					// namnv1104
					Monitor_Production.Pulse_In_2 := TRUE;
					Monitor_Production.Pulse_Out_2 := FALSE;
				END_IF
				// namnv - dieu kien tat tin hieu test vision
				IF GVL.Pro4_.Auto.Vs_On_Off  AND (GVL.Pro4_.Process.DATA_MC_VS = 1) THEN
					IF NOT GVL.Pro4_.Signal_In.T_Vs_detect.Q  THEN
						GVL.Pro4_.Auto.Vs_On_Off := FALSE;
						Pro_MC2_4 := 5;
						GVL.Pro4_.Process.DATA_TOOL_A1_IN_OLD := 0;
					ELSE
						//log
					END_IF
				ELSE
					Pro_MC2_4 := 5;
					GVL.Pro4_.Process.DATA_TOOL_A1_IN_OLD := 0;
				END_IF;
				
			END_IF
		40:	// Pick OK
			IF GVL.Pro4_.Process.DATA_TOOL_A2_OUT  = 2 AND Pick_A4_T2_Finish  THEN
				//GVL.Pro4_.Process.DATA_TOOL_A2_OUT := 2;
				Ton_OK_MC2_4.IN := FALSE;
				Ton_Limit_Test_VS.IN := FALSE;
				GVL.Pro4_.Process.DATA_MC_VS := 0;
				Pro_MC2_4 := 5;
			END_IF	
		50: // Pick NG
			IF GVL.Pro4_.Process.DATA_TOOL_A2_OUT  = 3 AND Pick_A4_T2_Finish  THEN
				//GVL.Pro4_.Process.DATA_TOOL_A2_OUT := 3;
				Ton_OK_MC2_4.IN := FALSE;
				Ton_Limit_Test_VS.IN := FALSE;
				GVL.Pro4_.Process.DATA_MC_VS := 0;
				Pro_MC2_4 := 5;
			END_IF
			
		60: // Pick NG - TS
			IF GVL.Pro4_.Process.DATA_TOOL_A2_OUT  = 4 AND Pick_A4_T2_Finish  THEN
				//GVL.Pro4_.Process.DATA_TOOL_A2_OUT := 3;
				Ton_OK_MC2_4.IN := FALSE;
				Ton_Limit_Test_VS.IN := FALSE;
				GVL.Pro4_.Process.DATA_MC_VS := 0;
				GVL.Pro4_.Process.DATA_TOOL_A1_IN_OLD := 0;
				Pro_MC2_4 := 5;
			END_IF
	END_CASE
END_ACTION

ACTION ACT_GO_Pos_Manual:
{region "1. GO HOME"}
Excute_Run_goHome_A := GVL.RB_A.Manual AND GVL.RB_A.RB_goHome_Comfirm AND GVL.RB_A_.Ready AND NOT GVL.RB_A_.Runing AND
					(GVL.RB_A.M1_goHome OR GVL.RB_A.M2_goHome OR GVL.RB_A.M3_goHome OR GVL.RB_A.M4_goHome );
Excute_Run_goHome_B := GVL.RB_B.Manual AND GVL.RB_B.RB_goHome_Comfirm AND GVL.RB_B_.Ready AND NOT GVL.RB_B_.Runing AND
					(GVL.RB_B.M1_goHome OR GVL.RB_B.M2_goHome OR GVL.RB_B.M3_goHome OR GVL.RB_B.M4_goHome );

IF GVL.RB_A.Manual AND GVL.RB_A.RB_goHome_Comfirm THEN
	GVL.RB_A.COORD := 0;
	IF GVL.RB_A.M1_goHome THEN Pos_run_manual_A.a.a0 := 0; ELSE Pos_run_manual_A.a.a0 := GVL.RB_A_.CUR_X ; END_IF;
	IF GVL.RB_A.M2_goHome THEN Pos_run_manual_A.a.a1 := 0; ELSE Pos_run_manual_A.a.a1 := GVL.RB_A_.CUR_Y ; END_IF;	
	IF GVL.RB_A.M3_goHome THEN Pos_run_manual_A.a.a2 := 0; ELSE Pos_run_manual_A.a.a2 := GVL.RB_A_.CUR_Z ; END_IF;	
	IF GVL.RB_A.M4_goHome THEN Pos_run_manual_A.a.a3 := 0; ELSE Pos_run_manual_A.a.a3 := GVL.RB_A_.CUR_R ; END_IF;	
END_IF

IF GVL.RB_B.Manual AND GVL.RB_B.RB_goHome_Comfirm THEN
	GVL.RB_B.COORD := 0;
	IF GVL.RB_B.M1_goHome THEN Pos_run_manual_B.a.a0 := 0; ELSE Pos_run_manual_B.a.a0 := GVL.RB_B_.CUR_X ; END_IF;	
	IF GVL.RB_B.M2_goHome THEN Pos_run_manual_B.a.a1 := 0; ELSE Pos_run_manual_B.a.a1 := GVL.RB_B_.CUR_Y ; END_IF;	
	IF GVL.RB_B.M3_goHome THEN Pos_run_manual_B.a.a2 := 0; ELSE Pos_run_manual_B.a.a2 := GVL.RB_B_.CUR_Z ; END_IF;	
	IF GVL.RB_B.M4_goHome THEN Pos_run_manual_B.a.a3 := 0; ELSE Pos_run_manual_B.a.a3 := GVL.RB_B_.CUR_R ; END_IF;
END_IF
{endregion}	

// Cai dat bien bao den vi tri muc tieu manual	 
IF (MOVP_A.Done OR MOVL_A.Done) 
AND (ABS(GVL.RB_A_.CUR_X - Pos_run_manual_A.c.X) < delta_position_cor) 
AND (ABS(GVL.RB_A_.CUR_Y - Pos_run_manual_A.c.Y) < delta_position_cor) 
AND (ABS(GVL.RB_A_.CUR_Z - Pos_run_manual_A.c.Z) < delta_position_cor) 
AND (ABS(GVL.RB_A_.CUR_R - Pos_run_manual_A.c.A) < delta_position_cor)
THEN  A_Comp_Man	:= TRUE;  ELSE A_Comp_Man	:= FALSE; END_IF;
IF (MOVP_B.Done OR MOVL_B.Done)  
AND (ABS(GVL.RB_B_.CUR_X - Pos_run_manual_B.c.X) < delta_position_cor) 
AND (ABS(GVL.RB_B_.CUR_Y - Pos_run_manual_B.c.Y) < delta_position_cor) 
AND (ABS(GVL.RB_B_.CUR_Z - Pos_run_manual_B.c.Z) < delta_position_cor) 
AND (ABS(GVL.RB_B_.CUR_R - Pos_run_manual_B.c.A) < delta_position_cor)
THEN  B_Comp_Man	:= TRUE;  ELSE B_Comp_Man	:= FALSE; END_IF;


{region "2. GO WAIT"}
// Jog & Teach
AP_Man_Z_Wait_Go := GVL.RB_A.Manual AND GVL.RB_A.Jog_Point AND GVL.RB_A.Move_Z_Wait AND GVL.RB_A_.Ready AND NOT GVL.RB_A_.Runing AND
						Pos_run_manual_A.c.Z = GVL_1.DATA_RB_A.Z_POS[1];
						IF GVL.RB_A.Move_Z_Wait AND POU_HMI_CONTROL_ROBOT.D_HMI_SCREEN = 21 THEN
							GVL.RB_A.COORD := 1;
							Pos_run_manual_A := POU_MONITOR_ROBOT.RB1_POS;
							Pos_run_manual_A.c.Z := GVL_1.DATA_RB_A.Z_POS[1];
						END_IF;																		
AP_Man_R_Wait_Go := GVL.RB_A.Manual AND GVL.RB_A.Jog_Point AND GVL.RB_A.Move_R_Wait AND GVL.RB_A_.Ready AND NOT GVL.RB_A_.Runing AND
						Pos_run_manual_A.c.A = GVL_1.DATA_RB_A.R_POS[1];
						IF GVL.RB_A.Move_R_Wait AND POU_HMI_CONTROL_ROBOT.D_HMI_SCREEN = 21 THEN
							GVL.RB_A.COORD := 1;
							Pos_run_manual_A := POU_MONITOR_ROBOT.RB1_POS;
							Pos_run_manual_A.c.A := GVL_1.DATA_RB_A.R_POS[1];
						END_IF;	
AP_Man_XY_Wait_Go := GVL.RB_A.Manual AND GVL.RB_A.Jog_Point AND GVL.RB_A.Move_XY_Wait AND GVL.RB_A_.Ready AND NOT GVL.RB_A_.Runing AND
						Pos_run_manual_A.c.X = GVL_1.DATA_RB_A.X_POS[1] AND Pos_run_manual_A.c.Y = GVL_1.DATA_RB_A.Y_POS[1] ;
						IF GVL.RB_A.Move_XY_Wait AND POU_HMI_CONTROL_ROBOT.D_HMI_SCREEN = 21 THEN
							GVL.RB_A.COORD := 1;
							Pos_run_manual_A := POU_MONITOR_ROBOT.RB1_POS;
							Pos_run_manual_A.c.X := GVL_1.DATA_RB_A.X_POS[1];
							Pos_run_manual_A.c.Y := GVL_1.DATA_RB_A.Y_POS[1];
						END_IF;	
/////////////////////////////////////////
Excute_Run_goZ_Wait_B := GVL.RB_B.Manual AND GVL.RB_B.Jog_Point AND GVL.RB_B.Move_Z_Wait AND GVL.RB_B_.Ready AND NOT GVL.RB_B_.Runing AND
						Pos_run_manual_B.c.Z = GVL_1.DATA_RB_B.Z_POS[1];
						IF GVL.RB_B.Move_Z_Wait AND POU_HMI_CONTROL_ROBOT.D_HMI_SCREEN = 31 THEN
							GVL.RB_B.COORD := 1;
							Pos_run_manual_B := POU_MONITOR_ROBOT.RB1_POS;
							Pos_run_manual_B.c.Z := GVL_1.DATA_RB_B.Z_POS[1];
						END_IF;																		
Excute_Run_goR_Wait_B := GVL.RB_B.Manual AND GVL.RB_B.Jog_Point AND GVL.RB_B.Move_R_Wait AND GVL.RB_B_.Ready AND NOT GVL.RB_B_.Runing AND
						Pos_run_manual_B.c.A = GVL_1.DATA_RB_B.R_POS[1];
						IF GVL.RB_B.Move_R_Wait AND POU_HMI_CONTROL_ROBOT.D_HMI_SCREEN = 31 THEN
							GVL.RB_B.COORD := 1;
							Pos_run_manual_B := POU_MONITOR_ROBOT.RB1_POS;
							Pos_run_manual_B.c.A := GVL_1.DATA_RB_B.R_POS[1];
						END_IF;	
Excute_Run_goXY_Wait_B := GVL.RB_B.Manual AND GVL.RB_B.Jog_Point AND GVL.RB_B.Move_XY_Wait AND GVL.RB_B_.Ready AND NOT GVL.RB_B_.Runing AND
						Pos_run_manual_B.c.X = GVL_1.DATA_RB_B.X_POS[1] AND Pos_run_manual_B.c.Y = GVL_1.DATA_RB_B.Y_POS[1] ;
						IF GVL.RB_B.Move_XY_Wait AND POU_HMI_CONTROL_ROBOT.D_HMI_SCREEN = 31 THEN
							GVL.RB_B.COORD := 1;
							Pos_run_manual_B := POU_MONITOR_ROBOT.RB1_POS;
							Pos_run_manual_B.c.X := GVL_1.DATA_RB_B.X_POS[1];
							Pos_run_manual_B.c.Y := GVL_1.DATA_RB_B.Y_POS[1];
						END_IF;	
{endregion}	
{region "3. GO SELECT POS"}
// ROBOT A
	AP_Man_Pos_Go := GVL.RB_A.Manual AND GVL.RB_A.Comfirm_Move AND GVL.RB_A_.Ready AND NOT GVL.RB_A_.Runing AND
							GVL.DW_[10] > 0 AND GVL.DW_[11] > 0 AND GVL.DW_[11] = 3;
	AP_Man_Pos_Go_L := GVL.RB_A.Manual AND GVL.RB_A.Comfirm_Move AND GVL.RB_A_.Ready AND NOT GVL.RB_A_.Runing AND
							GVL.DW_[10] > 0 AND GVL.DW_[11] > 0 AND GVL.DW_[11] = 1;
						IF GVL.RB_A.Comfirm_Move AND POU_HMI_CONTROL_ROBOT.D_HMI_SCREEN = 21 THEN
							GVL.RB_A.COORD := 1;						
							Pos_run_manual_A.c.X:= GVL_1.DATA_RB_A.X_POS[GVL.DW_[10]];
							Pos_run_manual_A.c.Y:= GVL_1.DATA_RB_A.Y_POS[GVL.DW_[10]];
							Pos_run_manual_A.c.Z:= GVL_1.DATA_RB_A.Z_POS[GVL.DW_[10]];
							Pos_run_manual_A.c.A:= GVL_1.DATA_RB_A.R_POS[GVL.DW_[10]];
							GVL.RB_A.Comfirm_Move := FALSE;											 
						END_IF;		
	Other_PosA := Pos_run_manual_A.c.X <> Pos_run_A_Pre.c.X OR Pos_run_manual_A.c.Y <> Pos_run_A_Pre.c.Y 
				  OR Pos_run_manual_A.c.Z <> Pos_run_A_Pre.c.Z OR Pos_run_manual_A.c.A <> Pos_run_A_Pre.c.A;	  											 
	Excute_Run_goPos_A_UpZ := GVL.RB_A.Manual AND GVL.RB_A.Comfirm_Up_Z AND GVL.RB_A_.Ready AND NOT GVL.RB_A_.Runing AND
							GVL.DW_[10] > 0 AND GVL.DW_[11] > 0;
	Excute_Run_goPos_A_UpZ_XY_BF_R := GVL.RB_A.Manual AND GVL.RB_A.Comfirm_Up_Z_XY_BF_R AND GVL.RB_A_.Ready AND NOT GVL.RB_A_.Runing AND
							GVL.DW_[10] > 0 AND GVL.DW_[11] > 0;
	Excute_Run_goPos_A_UpZ_R_BF_XY := GVL.RB_A.Manual AND GVL.RB_A.Comfirm_Up_Z_R_BF_XY AND GVL.RB_A_.Ready AND NOT GVL.RB_A_.Runing AND
							GVL.DW_[10] > 0 AND GVL.DW_[11] > 0;
						IF Excute_Run_goPos_A_UpZ AND POU_HMI_CONTROL_ROBOT.D_HMI_SCREEN = 21 THEN
							GVL.RB_A.COORD := 1;						
							RuningPosA[GVL.DW_[10]] := TRUE;
							mode_Run_GoPosA_manual := 1;	// chi len Z
							Pos_Run_A_Pre := Pos_0;		
							GVL.RB_A.Comfirm_Up_Z := FALSE; 
						ELSE
							IF Excute_Run_goPos_A_UpZ_XY_BF_R AND POU_HMI_CONTROL_ROBOT.D_HMI_SCREEN = 21 THEN
								GVL.RB_A.COORD := 1;						
								RuningPosA[GVL.DW_[10]] := TRUE;
								mode_Run_GoPosA_manual := 2;		// chay XY trc xoay R
								Pos_Run_A_Pre := Pos_0;		
								GVL.RB_A.Comfirm_Up_Z_XY_BF_R := FALSE;
							ELSE
								IF Excute_Run_goPos_A_UpZ_R_BF_XY AND POU_HMI_CONTROL_ROBOT.D_HMI_SCREEN = 21 THEN
									GVL.RB_A.COORD := 1;						
									RuningPosA[GVL.DW_[10]] := TRUE;
									mode_Run_GoPosA_manual := 3;		// xoay R trc XY
									Pos_Run_A_Pre := Pos_0;		
									GVL.RB_A.Comfirm_Up_Z_R_BF_XY := FALSE;
								END_IF; 
							END_IF;	 
						END_IF;	

IF NOT GVL.X[9] THEN
	RuningPosA[GVL.DW_[10]] := FALSE;
	RuningPosB[GVL.DW_[12]]	:= FALSE;	 
END_IF;
						 
IF RuningPosA[GVL.DW_[10]] THEN
	CASE PRO_A[GVL.DW_[10]] OF
			0: 
				Pos_run_manual_A :=  POU_MONITOR_ROBOT.RB1_POS;
				PRO_A[GVL.DW_[10]] := PRO_A[GVL.DW_[10]] + 10;
			10:
				Pos_run_manual_A.c.Z :=  GVL_1.DATA_RB_A.Z_POS[1];
				PRO_A[GVL.DW_[10]] := PRO_A[GVL.DW_[10]] + 10;
			20:
				IF Other_PosA THEN
					CASE GVL.DW_[11] OF
						1: 	excute_run_L_Upz_A := TRUE; 
						3:  AP_Man_UP_Z_Go := TRUE;
					END_CASE
					Pos_Run_A_Pre := Pos_run_manual_A; 
				END_IF
				IF GVL.RB_A_.ERROR OR  NOT GVL.RB_A_.Ready THEN
					RuningPosA[GVL.DW_[10]] := FALSE;
					excute_run_L_Upz_A := FALSE; 
					AP_Man_UP_Z_Go := FALSE;
			    END_IF
			    IF MOVL_A.Done OR MOVP_A.Done THEN
					excute_run_L_Upz_A := FALSE; 
					AP_Man_UP_Z_Go := FALSE;
					IF mode_Run_GoPosA_manual = 1 THEN
						PRO_A[GVL.DW_[10]] := PRO_A[GVL.DW_[10]] + 10;
					ELSE
						IF mode_Run_GoPosA_manual = 2 THEN
							PRO_A[GVL.DW_[10]] := PRO_A[GVL.DW_[10]] + 2;
						ELSE
							IF mode_Run_GoPosA_manual = 3 THEN
								PRO_A[GVL.DW_[10]] := PRO_A[GVL.DW_[10]] + 6;	 
							END_IF;
						END_IF;
					END_IF;
			    END_IF;
			22:
				Pos_run_manual_A.c.X :=  GVL_1.DATA_RB_A.X_POS[GVL.DW_[10]];
				Pos_run_manual_A.c.Y :=  GVL_1.DATA_RB_A.Y_POS[GVL.DW_[10]];	
				Pos_run_manual_A.c.Z :=  GVL.RB_A_.CUR_Z;					 
				Pos_run_manual_A.c.A :=  GVL.RB_A_.CUR_R;		  
				PRO_A[GVL.DW_[10]] := PRO_A[GVL.DW_[10]] + 2; 
			24:
				IF Other_PosA THEN
					CASE GVL.DW_[11] OF
						1: 	excute_run_L_Upz_A := TRUE; 
						3:  AP_Man_UP_Z_Go := TRUE;
					END_CASE
					Pos_Run_A_Pre := Pos_run_manual_A; 
				END_IF
				IF GVL.RB_A_.ERROR OR  NOT GVL.RB_A_.Ready THEN
					RuningPosA[GVL.DW_[10]] := FALSE;
					excute_run_L_Upz_A := FALSE; 
					AP_Man_UP_Z_Go := FALSE;
			    END_IF
			    IF MOVL_A.Done OR MOVP_A.Done THEN
					excute_run_L_Upz_A := FALSE; 
					AP_Man_UP_Z_Go := FALSE;
					PRO_A[GVL.DW_[10]] := 30;
			    END_IF	
			26:
				Pos_run_manual_A.c.X :=  GVL.RB_A_.CUR_X;
				Pos_run_manual_A.c.Y :=  GVL.RB_A_.CUR_Y;	
				Pos_run_manual_A.c.Z :=  GVL.RB_A_.CUR_Z;					 
				Pos_run_manual_A.c.A :=  GVL_1.DATA_RB_A.R_POS[GVL.DW_[10]];		  
				PRO_A[GVL.DW_[10]] := PRO_A[GVL.DW_[10]] + 2; 
			28:
				IF Other_PosA THEN
					CASE GVL.DW_[11] OF
						1: 	excute_run_L_Upz_A := TRUE; 
						3:  AP_Man_UP_Z_Go := TRUE;
					END_CASE
					Pos_Run_A_Pre := Pos_run_manual_A; 
				END_IF
				IF GVL.RB_A_.ERROR OR  NOT GVL.RB_A_.Ready THEN
					RuningPosA[GVL.DW_[10]] := FALSE;
					excute_run_L_Upz_A := FALSE; 
					AP_Man_UP_Z_Go := FALSE;
			    END_IF
			    IF MOVL_A.Done OR MOVP_A.Done THEN
					excute_run_L_Upz_A := FALSE; 
					AP_Man_UP_Z_Go := FALSE;
					PRO_A[GVL.DW_[10]] := 30;
			    END_IF 
			30:
				Pos_run_manual_A.c.X :=  GVL_1.DATA_RB_A.X_POS[GVL.DW_[10]];
				Pos_run_manual_A.c.Y :=  GVL_1.DATA_RB_A.Y_POS[GVL.DW_[10]];	
				Pos_run_manual_A.c.Z :=  GVL.RB_A_.CUR_Z;					 
				Pos_run_manual_A.c.A :=  GVL_1.DATA_RB_A.R_POS[GVL.DW_[10]];		  
				PRO_A[GVL.DW_[10]] := PRO_A[GVL.DW_[10]] + 10; 
			40:
				IF Other_PosA THEN
					CASE GVL.DW_[11] OF
						1: 	excute_run_L_Upz_A := TRUE; 
						3:  AP_Man_UP_Z_Go := TRUE;
					END_CASE
					Pos_Run_A_Pre := Pos_run_manual_A; 
				END_IF
				IF GVL.RB_A_.ERROR OR  NOT GVL.RB_A_.Ready THEN
					RuningPosA[GVL.DW_[10]] := FALSE;
					excute_run_L_Upz_A := FALSE; 
					AP_Man_UP_Z_Go := FALSE;
			    END_IF
			    IF MOVL_A.Done OR MOVP_A.Done THEN
					excute_run_L_Upz_A := FALSE; 
					AP_Man_UP_Z_Go := FALSE;
					PRO_A[GVL.DW_[10]] := PRO_A[GVL.DW_[10]] + 10;
			    END_IF	
			50:
				Pos_run_manual_A :=  POU_MONITOR_ROBOT.RB1_POS;
				PRO_A[GVL.DW_[10]] := PRO_A[GVL.DW_[10]] + 10;			 
			60:
				Pos_run_manual_A.c.Z :=  GVL_1.DATA_RB_A.Z_POS[GVL.DW_[10]];
				PRO_A[GVL.DW_[10]] := PRO_A[GVL.DW_[10]] + 10;
			70:
				IF Other_PosA THEN
					CASE GVL.DW_[11] OF
						1: 	excute_run_L_Upz_A := TRUE; 
						3:  AP_Man_UP_Z_Go := TRUE;
					END_CASE
					Pos_Run_A_Pre := Pos_run_manual_A; 
				END_IF
				IF GVL.RB_A_.ERROR OR  NOT GVL.RB_A_.Ready THEN
					RuningPosA[GVL.DW_[10]] := FALSE;
					excute_run_L_Upz_A := FALSE; 
					AP_Man_UP_Z_Go := FALSE;
			    END_IF
			    IF MOVL_A.Done OR MOVP_A.Done THEN
					excute_run_L_Upz_A := FALSE; 
					AP_Man_UP_Z_Go := FALSE;
					PRO_A[GVL.DW_[10]] := PRO_A[GVL.DW_[10]] + 10;
			    END_IF			  		   							 
											  
			80:/// HOÀN THÀNH ///  	   
					excute_run_L_Upz_A := FALSE; 
					AP_Man_UP_Z_Go := FALSE;
 			        RuningPosA[GVL.DW_[10]] := FALSE;				
					mode_Run_GoPosA_manual := 0; 
		 END_CASE
ELSE
	PRO_A[GVL.DW_[10]] := 0;	
	excute_run_L_Upz_A := FALSE; 
	AP_Man_UP_Z_Go := FALSE;
	mode_Run_GoPosA_manual := 0; 
END_IF;							  
// ROBOT B
	Excute_Run_goPos_B := GVL.RB_B.Manual AND GVL.RB_B.Comfirm_Move AND GVL.RB_B_.Ready AND NOT GVL.RB_B_.Runing AND
							GVL.DW_[12] > 0 AND GVL.DW_[13] > 0 AND GVL.DW_[13] = 3;
	Excute_Run_goPos_B_L := GVL.RB_B.Manual AND GVL.RB_B.Comfirm_Move AND GVL.RB_B_.Ready AND NOT GVL.RB_B_.Runing AND
							GVL.DW_[12] > 0 AND GVL.DW_[13] > 0 AND GVL.DW_[13] = 1;
							
						IF GVL.RB_B.Comfirm_Move AND POU_HMI_CONTROL_ROBOT.D_HMI_SCREEN = 31 THEN
							GVL.RB_B.COORD := 1;						
							Pos_run_manual_B.c.X:= GVL_1.DATA_RB_B.X_POS[GVL.DW_[12]];
							Pos_run_manual_B.c.Y:= GVL_1.DATA_RB_B.Y_POS[GVL.DW_[12]];
							Pos_run_manual_B.c.Z:= GVL_1.DATA_RB_B.Z_POS[GVL.DW_[12]];
							Pos_run_manual_B.c.A:= GVL_1.DATA_RB_B.R_POS[GVL.DW_[12]];
							GVL.RB_B.Comfirm_Move := FALSE;											 
						END_IF;		
	Other_PosB := Pos_run_manual_B.c.X <> Pos_Run_B_Pre.c.X OR Pos_run_manual_B.c.Y <> Pos_Run_B_Pre.c.Y 
				  OR Pos_run_manual_B.c.Z <> Pos_Run_B_Pre.c.Z OR Pos_run_manual_B.c.A <> Pos_Run_B_Pre.c.A;	  											 
	Excute_Run_goPos_B_UpZ := GVL.RB_B.Manual AND GVL.RB_B.Comfirm_Up_Z AND GVL.RB_B_.Ready AND NOT GVL.RB_B_.Runing AND
							GVL.DW_[12] > 0 AND GVL.DW_[13] > 0;
	Excute_Run_goPos_B_UpZ_XY_BF_R := GVL.RB_B.Manual AND GVL.RB_B.Comfirm_Up_Z_XY_BF_R AND GVL.RB_B_.Ready AND NOT GVL.RB_B_.Runing AND
							GVL.DW_[12] > 0 AND GVL.DW_[13] > 0;
	Excute_Run_goPos_B_UpZ_R_BF_XY := GVL.RB_B.Manual AND GVL.RB_B.Comfirm_Up_Z_R_BF_XY AND GVL.RB_B_.Ready AND NOT GVL.RB_B_.Runing AND
							GVL.DW_[12] > 0 AND GVL.DW_[13] > 0;
						IF Excute_Run_goPos_B_UpZ AND POU_HMI_CONTROL_ROBOT.D_HMI_SCREEN = 31 THEN
							GVL.RB_B.COORD := 1;						
							RuningPosB[GVL.DW_[12]] := TRUE;
							mode_Run_GoPosB_manual := 1;	
							Pos_Run_B_Pre := Pos_0;	
							GVL.RB_B.Comfirm_Up_Z := FALSE;
						ELSE
							IF Excute_Run_goPos_B_UpZ_XY_BF_R AND POU_HMI_CONTROL_ROBOT.D_HMI_SCREEN = 31 THEN
								GVL.RB_B.COORD := 1;						
								RuningPosB[GVL.DW_[12]] := TRUE;
								mode_Run_GoPosB_manual := 2;	
								Pos_Run_B_Pre := Pos_0;	
								GVL.RB_B.Comfirm_Up_Z_XY_BF_R := FALSE;	 
							ELSE
								IF Excute_Run_goPos_B_UpZ_R_BF_XY AND POU_HMI_CONTROL_ROBOT.D_HMI_SCREEN = 31 THEN
									GVL.RB_B.COORD := 1;						
									RuningPosB[GVL.DW_[12]] := TRUE;
									mode_Run_GoPosB_manual := 3;	
									Pos_Run_B_Pre := Pos_0;	
									GVL.RB_B.Comfirm_Up_Z_R_BF_XY := FALSE;
								 END_IF;
							END_IF;
						END_IF;							 
IF RuningPosB[GVL.DW_[12]] THEN
	CASE PRO_B[GVL.DW_[12]] OF
			0: 
				Pos_run_manual_B :=  POU_MONITOR_ROBOT.RB2_POS;
				PRO_B[GVL.DW_[12]] := PRO_B[GVL.DW_[12]] + 10;
			10:
				Pos_run_manual_B.c.Z :=  GVL_1.DATA_RB_B.Z_POS[1];
				PRO_B[GVL.DW_[12]] := PRO_B[GVL.DW_[12]] + 10;
			20:
				IF Other_PosB THEN
					CASE GVL.DW_[13] OF
						1: 	excute_run_L_Upz_B := TRUE; 
						3:  excute_run_P_Upz_B := TRUE;
					END_CASE
					Pos_Run_B_Pre := Pos_run_manual_B; 
				END_IF
				IF GVL.RB_B_.ERROR OR  NOT GVL.RB_B_.Ready THEN
					RuningPosB[GVL.DW_[12]] := FALSE;
					excute_run_L_Upz_B := FALSE; 
					excute_run_P_Upz_B := FALSE;
			    END_IF
			    IF MOVL_B.Done OR MOVP_B.Done THEN
					excute_run_L_Upz_B := FALSE; 
					excute_run_P_Upz_B := FALSE;
					IF mode_Run_GoPosB_manual = 1 THEN
						PRO_B[GVL.DW_[12]] := PRO_B[GVL.DW_[12]] + 10;
					ELSE
						IF mode_Run_GoPosB_manual = 2 THEN
							PRO_B[GVL.DW_[12]] := PRO_B[GVL.DW_[12]] + 2;
						ELSE
							IF mode_Run_GoPosB_manual = 3 THEN
								PRO_B[GVL.DW_[12]] := PRO_B[GVL.DW_[12]] + 6;	 
							END_IF;
						END_IF;
					END_IF;
			    END_IF
			22:
				Pos_run_manual_B.c.X :=  GVL_1.DATA_RB_B.X_POS[GVL.DW_[12]];
				Pos_run_manual_B.c.Y :=  GVL_1.DATA_RB_B.Y_POS[GVL.DW_[12]];	
				Pos_run_manual_B.c.Z :=  GVL.RB_B_.CUR_Z;					 
				Pos_run_manual_B.c.A :=  GVL.RB_B_.CUR_R;		  
				PRO_B[GVL.DW_[12]] := PRO_B[GVL.DW_[12]] + 2;  
			24:
				IF Other_PosB THEN
					CASE GVL.DW_[13] OF
						1: 	excute_run_L_Upz_B := TRUE; 
						3:  excute_run_P_Upz_B := TRUE;
					END_CASE
					Pos_Run_B_Pre := Pos_run_manual_B; 
				END_IF
				IF GVL.RB_B_.ERROR OR NOT GVL.RB_B_.Ready THEN
					RuningPosB[GVL.DW_[12]] := FALSE;
					excute_run_L_Upz_B := FALSE; 
					excute_run_P_Upz_B := FALSE;
			    END_IF
			    IF MOVL_B.Done OR MOVP_B.Done THEN
					excute_run_L_Upz_B := FALSE; 
					excute_run_P_Upz_B := FALSE;
					PRO_B[GVL.DW_[12]] := 30;
			    END_IF
			26:
				Pos_run_manual_B.c.X :=  GVL.RB_B_.CUR_X;
				Pos_run_manual_B.c.Y :=  GVL.RB_B_.CUR_Y;	
				Pos_run_manual_B.c.Z :=  GVL.RB_B_.CUR_Z;					 
				Pos_run_manual_B.c.A :=  GVL_1.DATA_RB_B.r_POS[GVL.DW_[12]];		  
				PRO_B[GVL.DW_[12]] := PRO_B[GVL.DW_[12]] + 2;
			28:
				IF Other_PosB THEN
					CASE GVL.DW_[13] OF
						1: 	excute_run_L_Upz_B := TRUE; 
						3:  excute_run_P_Upz_B := TRUE;
					END_CASE
					Pos_Run_B_Pre := Pos_run_manual_B; 
				END_IF
				IF GVL.RB_B_.ERROR OR NOT GVL.RB_B_.Ready THEN
					RuningPosB[GVL.DW_[12]] := FALSE;
					excute_run_L_Upz_B := FALSE; 
					excute_run_P_Upz_B := FALSE;
			    END_IF
			    IF MOVL_B.Done OR MOVP_B.Done THEN
					excute_run_L_Upz_B := FALSE; 
					excute_run_P_Upz_B := FALSE;
					PRO_B[GVL.DW_[12]] := 30;
			    END_IF 
			30:
				Pos_run_manual_B.c.X :=  GVL_1.DATA_RB_B.X_POS[GVL.DW_[12]];
				Pos_run_manual_B.c.Y :=  GVL_1.DATA_RB_B.Y_POS[GVL.DW_[12]];	
				Pos_run_manual_B.c.Z :=  GVL.RB_B_.CUR_Z;					 
				Pos_run_manual_B.c.A :=  GVL_1.DATA_RB_B.r_POS[GVL.DW_[12]];		  
				PRO_B[GVL.DW_[12]] := PRO_B[GVL.DW_[12]] + 10; 
			40:
				IF Other_PosB THEN
					CASE GVL.DW_[13] OF
						1: 	excute_run_L_Upz_B := TRUE; 
						3:  excute_run_P_Upz_B := TRUE;
					END_CASE
					Pos_Run_B_Pre := Pos_run_manual_B; 
				END_IF
				IF GVL.RB_B_.ERROR OR NOT GVL.RB_B_.Ready THEN
					RuningPosB[GVL.DW_[12]] := FALSE;
					excute_run_L_Upz_B := FALSE; 
					excute_run_P_Upz_B := FALSE;
			    END_IF
			    IF MOVL_B.Done OR MOVP_B.Done THEN
					excute_run_L_Upz_B := FALSE; 
					excute_run_P_Upz_B := FALSE;
					PRO_B[GVL.DW_[12]] := PRO_B[GVL.DW_[12]] + 10;
			    END_IF
			50:
				Pos_run_manual_B :=  POU_MONITOR_ROBOT.RB2_POS;
				PRO_B[GVL.DW_[12]] := PRO_B[GVL.DW_[12]] + 10;			 
			60:
				Pos_run_manual_B.c.Z :=  GVL_1.DATA_RB_B.Z_POS[GVL.DW_[12]];
				PRO_B[GVL.DW_[12]] := PRO_B[GVL.DW_[12]] + 10;
			70:
				IF Other_PosB THEN
					CASE GVL.DW_[13] OF
						1: 	excute_run_L_Upz_B := TRUE; 
						3:  excute_run_P_Upz_B := TRUE;
					END_CASE
					Pos_Run_B_Pre := Pos_run_manual_B; 
				END_IF
				IF GVL.RB_B_.ERROR OR  NOT GVL.RB_b_.Ready THEN
					RuningPosB[GVL.DW_[12]] := FALSE;
					excute_run_L_Upz_B := FALSE; 
					excute_run_P_Upz_B := FALSE;
			    END_IF
			    IF MOVL_B.Done OR MOVP_B.Done THEN
					excute_run_L_Upz_B := FALSE; 
					excute_run_P_Upz_B := FALSE;
					PRO_B[GVL.DW_[12]] := PRO_B[GVL.DW_[12]] + 10;
			    END_IF	
			80:/// HOÀN THÀNH ///  	   
					excute_run_L_Upz_B := FALSE; 
					excute_run_P_Upz_B := FALSE;
 			        RuningPosB[GVL.DW_[12]] := FALSE;			
					mode_Run_GoPosB_manual := 0;	 
		 END_CASE
ELSE
	PRO_B[GVL.DW_[12]] := 0;	
	excute_run_L_Upz_b := FALSE; 
	excute_run_P_Upz_b := FALSE;		
	mode_Run_GoPosB_manual := 0;	 
END_IF;										   
{endregion}	
	 
{region "4. Pos Cam"}	 
// excute_run_cam_B := GVL.RB_B.Manual AND GVL.RB_B_.Ready AND NOT GVL.RB_B_.Runing AND GVL.RB_B.move_Pos_cam ;
// 	 					 
// 						IF GVL.RB_B.move_Pos_cam AND POU_HMI_CONTROL_ROBOT.D_HMI_SCREEN = 31 THEN
// 							GVL.RB_B.COORD := 1;
// 							Pos_run_manual_B := POU_MONITOR_ROBOT.RB1_POS;
// 							Pos_run_manual_B.c.X := GVL_1.DATA_RB_B.X_POS[1];
// 							Pos_run_manual_B.c.Y := GVL_1.DATA_RB_B.Y_POS[1];
// 						END_IF;		  
// ROBOT B
	excute_run_cam_B := GVL.RB_B.Manual AND GVL.RB_B_.Ready AND NOT GVL.RB_B_.Runing AND GVL.RB_B.move_Pos_cam ;	
	  											 
						IF excute_run_cam_B AND POU_HMI_CONTROL_ROBOT.D_HMI_SCREEN = 181 THEN
							GVL.RB_B.COORD := 1;						
							Running_B_Cam := TRUE;	
							Pos_Run_B_Pre := Pos_0;	
							excute_run_cam_B := FALSE;	 
						END_IF;							 
IF Running_B_Cam THEN
	CASE Pro_B_cam OF
			0: 
				Pos_run_manual_B :=  POU_MONITOR_ROBOT.RB2_POS;
				Pro_B_cam := Pro_B_cam + 10;
			10:
				Pos_run_manual_B.c.Z :=  GVL_1.DATA_RB_B.Z_POS[1];
				Pro_B_cam := Pro_B_cam + 10;
			20:
				IF Other_PosB THEN
				excute_run_P_cam_B := TRUE;
				Pos_Run_B_Pre := Pos_run_manual_B; 
				END_IF;
				IF GVL.RB_B_.ERROR OR  NOT GVL.RB_B_.Ready THEN
					excute_run_P_cam_B := FALSE;
				    Running_B_Cam := FALSE;
			    END_IF
			    IF MOVP_B.Done THEN
					excute_run_P_cam_B := FALSE;
					Pro_B_cam := Pro_B_cam + 10;
			    END_IF
			30:
				CASE GVL.DW_[20] OF
					0:
						Pos_run_manual_B.c.X :=  GVL.Cam_T1.POS_X_RESULT;
						Pos_run_manual_B.c.Y :=  GVL.Cam_T1.POS_Y_RESULT;	  					 
					1:	 
						Pos_run_manual_B.c.X :=  GVL.Cam_T2.POS_X_RESULT;
						Pos_run_manual_B.c.Y :=  GVL.Cam_T2.POS_Y_RESULT;	 
				END_CASE		  
						Pos_run_manual_B.c.Z :=  GVL.RB_B_.CUR_Z;					 
						Pos_run_manual_B.c.A :=  GVL_1.DATA_RB_B.r_POS[1];					   
				Pro_B_cam := Pro_B_cam + 10;
			40:
				IF Other_PosB THEN
				excute_run_P_cam_B := TRUE;
				Pos_Run_B_Pre := Pos_run_manual_B; 
				END_IF;
				IF GVL.RB_B_.ERROR OR  NOT GVL.RB_B_.Ready THEN
					excute_run_P_cam_B := FALSE;
				    Running_B_Cam := FALSE;
			    END_IF
			    IF MOVP_B.Done THEN
					excute_run_P_cam_B := FALSE;
					Pro_B_cam := Pro_B_cam + 10;
			    END_IF			 
			50:
				GVL.RB_B.COORD := 1;
				Pos_run_manual_B :=  POU_MONITOR_ROBOT.RB2_POS;
				Pro_B_cam := Pro_B_cam + 10;		 
			60:
				Pos_run_manual_B.c.Z :=  GVL_1.DATA_RB_B.Z_POS[1];
				Pro_B_cam := Pro_B_cam + 10;
			70:
				IF Other_PosB THEN
				excute_run_P_cam_B := TRUE;
				Pos_Run_B_Pre := Pos_run_manual_B; 
				END_IF;
				IF GVL.RB_B_.ERROR OR  NOT GVL.RB_B_.Ready THEN
					excute_run_P_cam_B := FALSE;
				    Running_B_Cam := FALSE;
			    END_IF
			    IF MOVP_B.Done THEN
					excute_run_P_cam_B := FALSE;
					Pro_B_cam := Pro_B_cam + 10;
			    END_IF
			80:/// HOÀN THÀNH ///  	   
					excute_run_P_cam_B:= FALSE; 
 			        Running_B_Cam := FALSE;				 
		 END_CASE
ELSE
	Pro_B_cam := 0;	 
	excute_run_P_cam_B := FALSE;		 
END_IF;			   
/// Test Pick by Cam						
	  											 
IF GVL.MB_[11]  THEN
	CASE Test_Pick OF
			0: 
				Pos_run_manual_B :=  POU_MONITOR_ROBOT.RB2_POS;
				Test_Pick := Test_Pick + 10;
			10:
				Pos_run_manual_B.c.Z :=  GVL_1.DATA_RB_B.Z_POS[1];
				Test_Pick := Test_Pick + 10;
			20:
				IF Other_PosB THEN
				run_P_cam_B_test_pick := TRUE;
				Pos_Run_B_Pre := Pos_run_manual_B; 
				END_IF;
				IF GVL.RB_B_.ERROR OR  NOT GVL.RB_B_.Ready THEN
					run_P_cam_B_test_pick := FALSE;
				    GVL.MB_[11] := FALSE;
			    END_IF
			    IF MOVP_B.Done THEN
					run_P_cam_B_test_pick := FALSE;
					Test_Pick := Test_Pick + 10;
			    END_IF
			30:
				 CASE GVL.DW_[20] OF
					0:
						Pos_run_manual_B.c.X :=  GVL.Cam_T1.POS_X_RESULT;
						Pos_run_manual_B.c.Y :=  GVL.Cam_T1.POS_Y_RESULT;					
					1:	  
						Pos_run_manual_B.c.X :=  GVL.Cam_T2.POS_X_RESULT;
						Pos_run_manual_B.c.Y :=  GVL.Cam_T2.POS_Y_RESULT;						 							  
				 END_CASE	  
				Pos_run_manual_B.c.Z :=  GVL.RB_B_.CUR_Z;					 
				Pos_run_manual_B.c.A :=  GVL_1.DATA_RB_B.r_POS[1];	
// 					 IF GVL.Cam_T2.POS_R_RESULT < 180 THEN
// 						Pos_run_manual_B.c.A:= GVL_1.DATA_RB_B.R_POS[1] + GVL.Cam_T2.POS_R_RESULT ;	  
// 					ELSE
// 						Pos_run_manual_B.c.A:= GVL_1.DATA_RB_B.R_POS[1] - (360-GVL.Cam_T2.POS_R_RESULT) ;	 
// 					END_IF	  
				Test_Pick := Test_Pick + 10;
			40:
				IF Other_PosB THEN
				run_P_cam_B_test_pick := TRUE;
				Pos_Run_B_Pre := Pos_run_manual_B; 
				END_IF;
				IF GVL.RB_B_.ERROR OR  NOT GVL.RB_B_.Ready THEN
					run_P_cam_B_test_pick := FALSE;
				    GVL.MB_[11] := FALSE;
			    END_IF
			    IF MOVP_B.Done THEN
					run_P_cam_B_test_pick := FALSE;
					Test_Pick := Test_Pick + 10;
			    END_IF
			50:
				Pos_run_manual_B :=  POU_MONITOR_ROBOT.RB2_POS;
				Test_Pick := Test_Pick + 10;		 
			60:
				Pos_run_manual_B.c.Z :=  GVL_1.DATA_RB_B.Z_POS[1];
				Test_Pick := Test_Pick + 10;
			70:
				IF Other_PosB THEN
				run_P_cam_B_test_pick := TRUE;
				Pos_Run_B_Pre := Pos_run_manual_B; 
				END_IF;
				IF GVL.RB_B_.ERROR OR  NOT GVL.RB_B_.Ready THEN
					run_P_cam_B_test_pick := FALSE;
				    GVL.MB_[11] := FALSE;
			    END_IF
			    IF MOVP_B.Done THEN
					run_P_cam_B_test_pick := FALSE;
					Test_Pick := Test_Pick + 10;
			    END_IF
			80:	
				 CASE GVL.RB_B.Number_Tool OF
					1:
						GVL.RB_B.Vacuum_1 := TRUE;				
					2:	  
						GVL.RB_B.Vacuum_2 := TRUE;						 							  
				 END_CASE					 
					//Project_3_Delay_A(IN:= TRUE, PT := T#500MS);
				IF Project_3_Delay_A.Q THEN
					Test_Pick := Test_Pick + 10;	
				END_IF;						  
			90: 
				Project_3_Delay_A.IN	:= FALSE;
				Pos_run_manual_B :=  POU_MONITOR_ROBOT.RB2_POS;
				Test_Pick := Test_Pick + 10;
			100:
				Pos_run_manual_B.c.Z :=  GVL_1.DATA_RB_B.Z_POS[1];
				Test_Pick := Test_Pick + 10;
			110:
				IF Other_PosB THEN
				run_P_cam_B_test_pick := TRUE;
				Pos_Run_B_Pre := Pos_run_manual_B; 
				END_IF;
				IF GVL.RB_B_.ERROR OR  NOT GVL.RB_B_.Ready THEN
					run_P_cam_B_test_pick := FALSE;
				    GVL.MB_[11] := FALSE;
			    END_IF
			    IF MOVP_B.Done THEN
					run_P_cam_B_test_pick := FALSE;
					Test_Pick := Test_Pick + 10;
			    END_IF	
			120:
				Pos_run_manual_B.c.X:= GVL_1.DATA_RB_B.X_POS[1];
				Pos_run_manual_B.c.Y:= GVL_1.DATA_RB_B.Y_POS[1];
				Pos_run_manual_B.c.Z:= GVL.RB_B_.CUR_Z;
				Pos_run_manual_B.c.A:= GVL_1.DATA_RB_B.R_POS[1];				 
				Test_Pick := Test_Pick + 10;
			130:
				IF Other_PosB THEN
				run_P_cam_B_test_pick := TRUE;
				Pos_Run_B_Pre := Pos_run_manual_B; 
				END_IF;
				IF GVL.RB_B_.ERROR OR  NOT GVL.RB_B_.Ready THEN
					run_P_cam_B_test_pick := FALSE;
				    GVL.MB_[11] := FALSE;
			    END_IF
			    IF MOVP_B.Done THEN
					run_P_cam_B_test_pick := FALSE;
					Test_Pick := Test_Pick + 10;
			    END_IF						   
			140:/// HOÀN THÀNH ///  	   
					run_P_cam_B_test_pick:= FALSE; 
 			        GVL.MB_[11] := FALSE;			 
		 END_CASE	 
ELSE
run_P_cam_B_test_pick:= FALSE;		 
Test_Pick := 0;			  
END_IF;							 

IF GVL.MB_[12]  THEN
	CASE Test_Place OF
			0: 
				Pos_run_manual_B :=  POU_MONITOR_ROBOT.RB2_POS;
				test_Place := test_Place + 10;
			10:
				Pos_run_manual_B.c.Z :=  GVL_1.DATA_RB_B.Z_POS[1];
				test_Place := test_Place + 10;
			20:
				IF Other_PosB THEN
				run_P_cam_B_test_Place := TRUE;
				Pos_Run_B_Pre := Pos_run_manual_B; 
				END_IF;
				IF GVL.RB_B_.ERROR OR  NOT GVL.RB_B_.Ready THEN
					run_P_cam_B_test_Place := FALSE;
				    GVL.MB_[12] := FALSE;
			    END_IF
			    IF MOVP_B.Done THEN
					run_P_cam_B_test_Place := FALSE;
					test_Place := test_Place + 10;
			    END_IF
			30:
				Pos_run_manual_B.c.X:= GVL_1.DATA_RB_B.X_POS[2];
				Pos_run_manual_B.c.Y:= GVL_1.DATA_RB_B.Y_POS[2];
				Pos_run_manual_B.c.Z:= GVL.RB_B_.CUR_Z;
				Pos_run_manual_B.c.A:= GVL_1.DATA_RB_B.R_POS[2];	 
// 				 CASE GVL.DW_[20] OF
// 					0:
// 						 IF GVL.Cam_T1.POS_R_RESULT < 0 THEN
// 							Pos_run_manual_B.c.A:= GVL_1.DATA_RB_B.R_POS[2] - GVL.Cam_T1.POS_R_RESULT ;	  
// 						ELSE
// 							Pos_run_manual_B.c.A:= GVL_1.DATA_RB_B.R_POS[2] + GVL.Cam_T1.POS_R_RESULT ;	 
// 						END_IF					
// 					1:	  
// 						 IF GVL.Cam_T2.POS_R_RESULT < 0 THEN
// 							Pos_run_manual_B.c.A:= GVL_1.DATA_RB_B.R_POS[2] - GVL.Cam_T2.POS_R_RESULT ;	  
// 						ELSE
// 							Pos_run_manual_B.c.A:= GVL_1.DATA_RB_B.R_POS[2] + GVL.Cam_T2.POS_R_RESULT ;	 
// 						END_IF						 							  
// 				 END_CASE					  
				test_Place := test_Place + 10;
			40:
				IF Other_PosB THEN
				run_P_cam_B_test_Place := TRUE;
				Pos_Run_B_Pre := Pos_run_manual_B; 
				END_IF;
				IF GVL.RB_B_.ERROR OR  NOT GVL.RB_B_.Ready THEN
					run_P_cam_B_test_Place := FALSE;
				    GVL.MB_[12] := FALSE;
			    END_IF
			    IF MOVP_B.Done THEN
					run_P_cam_B_test_Place := FALSE;
					test_Place := test_Place + 1;
			    END_IF
			41:
				 CASE GVL.DW_[20] OF
					0:
						 IF GVL.Cam_T1.POS_R_RESULT < 0 THEN
							Pos_run_manual_B.c.A:=  GVL_1.DATA_RB_B.R_POS[2] + GVL.Cam_T1.POS_R_RESULT ;	  
							test_Place := test_Place + 1;	 
						ELSE
							Pos_run_manual_B.c.A:=  GVL_1.DATA_RB_B.R_POS[2] - GVL.Cam_T1.POS_R_RESULT ;	
 							test_Place := test_Place + 1;
						END_IF					
					1:	  
						 IF GVL.Cam_T2.POS_R_RESULT < 0 THEN
							Pos_run_manual_B.c.A:=  GVL_1.DATA_RB_B.R_POS[2] + GVL.Cam_T2.POS_R_RESULT ;
							test_Place := test_Place + 1;
  
						ELSE
							Pos_run_manual_B.c.A:=  GVL_1.DATA_RB_B.R_POS[2] - GVL.Cam_T2.POS_R_RESULT ;
							test_Place := test_Place + 1;	 
						END_IF						 							  
				 END_CASE					 
			42:
				IF Other_PosB THEN
				run_P_cam_B_test_Place := TRUE;
				Pos_Run_B_Pre := Pos_run_manual_B; 
				END_IF;
				IF GVL.RB_B_.ERROR OR  NOT GVL.RB_B_.Ready THEN
					run_P_cam_B_test_Place := FALSE;
				    GVL.MB_[12] := FALSE;
			    END_IF
			    IF MOVP_B.Done THEN
					run_P_cam_B_test_Place := FALSE;
					test_Place := 50;
			    END_IF				 
					  
			50:
				Pos_run_manual_B :=  POU_MONITOR_ROBOT.RB2_POS;
				test_Place := test_Place + 10;		 
			60:
				Pos_run_manual_B.c.Z :=  GVL_1.DATA_RB_B.Z_POS[2];
				test_Place := test_Place + 10;
			70:
				IF Other_PosB THEN
				run_P_cam_B_test_Place := TRUE;
				Pos_Run_B_Pre := Pos_run_manual_B; 
				END_IF;
				IF GVL.RB_B_.ERROR OR  NOT GVL.RB_B_.Ready THEN
					run_P_cam_B_test_Place := FALSE;
				    GVL.MB_[12] := FALSE;
			    END_IF
			    IF MOVP_B.Done THEN
					run_P_cam_B_test_Place := FALSE;
					test_Place := test_Place + 10;
			    END_IF
			80:		 
				CASE GVL.RB_B.Number_Tool OF
					0:
						GVL.RB_B.Vacuum_1 := FALSE; 
						GVL.RB_B.Vacuum_2 := FALSE;	 
					1: 	 			
						GVL.RB_B.Vacuum_1 := FALSE;
					2:
						GVL.RB_B.Vacuum_2 := FALSE; 
				END_CASE
					Project_3_Delay_B(IN:= TRUE, PT := T#500MS);
				IF Project_3_Delay_B.Q THEN
					test_Place := test_Place + 10;	
				END_IF;						  
			90: 
				Project_3_Delay_B.IN	:= FALSE;
				Pos_run_manual_B :=  POU_MONITOR_ROBOT.RB2_POS;
				test_Place := test_Place + 10;
			100:
				Pos_run_manual_B.c.Z :=  GVL_1.DATA_RB_B.Z_POS[1];
				test_Place := test_Place + 10;
			110:
				IF Other_PosB THEN
				run_P_cam_B_test_Place := TRUE;
				Pos_Run_B_Pre := Pos_run_manual_B; 
				END_IF;
				IF GVL.RB_B_.ERROR OR  NOT GVL.RB_B_.Ready THEN
					run_P_cam_B_test_Place := FALSE;
				    GVL.MB_[12] := FALSE;
			    END_IF
			    IF MOVP_B.Done THEN
					run_P_cam_B_test_Place := FALSE;
					test_Place := test_Place + 10;
			    END_IF	
			120:
				Pos_run_manual_B.c.X:= GVL_1.DATA_RB_B.X_POS[1];
				Pos_run_manual_B.c.Y:= GVL_1.DATA_RB_B.Y_POS[1];
				Pos_run_manual_B.c.Z:= GVL.RB_B_.CUR_Z;
				Pos_run_manual_B.c.A:= GVL_1.DATA_RB_B.R_POS[1];				 
				test_Place := test_Place + 10;
			130:
				IF Other_PosB THEN
				run_P_cam_B_test_Place := TRUE;
				Pos_Run_B_Pre := Pos_run_manual_B; 
				END_IF;
				IF GVL.RB_B_.ERROR OR  NOT GVL.RB_B_.Ready THEN
					run_P_cam_B_test_Place := FALSE;
				    GVL.MB_[12] := FALSE;
			    END_IF
			    IF MOVP_B.Done THEN
					run_P_cam_B_test_Place := FALSE;
					test_Place := test_Place + 10;
			    END_IF						   
			140:/// HOÀN THÀNH ///  	   
					run_P_cam_B_test_Place:= FALSE; 
 			        GVL.MB_[12] := FALSE;			 
		 END_CASE	 
ELSE
run_P_cam_B_test_Place:= FALSE;		 
test_Place := 0;			  
END_IF;	

// Chu trinh calib project 4	 
// Off_Calib_FtrigB(CLK := GVL.Pro4_.Man.Run_Calib_Pos);
// IF ((i_Vs_Align = 12) AND (GVL.Pro4_.Man.Result_Calib_Done OR GVL.Pro4_.Man.Result_Trigger_Vs_Align_Done)) OR Off_Calib_FtrigB.Q THEN
// 		i_Vs_Align := 0;
// 		GVL.Pro4_.Man.Run_Calib_Pos := FALSE;
// 		Calib_first_bit := FALSE;
// 		GVL.Pro4_.Man.Lighting_On_Off := FALSE;
// 		GVL.Pro4_.Man.Run_Calib_Pos_Done := FALSE;
// 		T_Delay_Trigger_Calib.IN := FALSE;
// 		GVL.Pro4_.Man.Trigger_Vs_Align_On_Off := FALSE;
// 		Run_One_Pos_Calib := FALSE;
// END_IF
// IF (GVL.Pro4_.Man.Run_Calib_Pos) THEN
// 	IF (NOT Calib_first_bit) THEN
// 		FOR i_Vs_Align_old := 16 TO 87 BY 1 DO
// 			GVL.MODBUS[i_Vs_Align_old] := 0;	 
// 		END_FOR
// 		i_Vs_Align := 0;
// 		Calib_first_bit := TRUE;
// 		GVL.Pro4_.Man.Result_Trigger_Vs_Align_Done := FALSE;
// 		Run_One_Pos_Calib := FALSE;
// 		GVL.Pro4_.Man.Lighting_On_Off := TRUE;
// 	END_IF
// 	B_Auto_Calib_4();
// END_IF
Robot_Calib_Vision();
							  
{endregion}
END_ACTION

ACTION B_Auto_Calib_4:
Trigger_Calib_Done(CLK := GVL.Pro4_.Man.Result_Trigger_Vs_Align_Done);
T_Delay_Trigger_Calib(PT := TO_TIME(GVL.Pro4_.ST_MC.Delay_Trigger_Vision_Align)*100);
//WHILE i_Vs_Align < 12 AND GVL.Pro4_.Man.Run_Calib_Pos DO
M_CHOOSE_POS_Man(DATA := 1, ID := i_Vs_Align + 34, XYR_CONST := FALSE, Z_CONST:= FALSE); // pos 2
IF NOT excute_run_P_cam_B AND NOT Run_One_Pos_Calib THEN
	// B_Comp := FALSE;
	excute_run_P_cam_B := TRUE;
END_IF		
IF MOVP_B.Error OR MOVL_B.Error THEN
	excute_run_P_cam_B	:= FALSE;	 	 
END_IF;				
IF MOVP_B.Done AND excute_run_P_cam_B THEN
	Run_One_Pos_Calib := TRUE;
	excute_run_P_cam_B :=FALSE;	
	T_Delay_Trigger_Calib.IN := TRUE;
	GVL.Pro4_.Man.Trigger_Vs_Align_On_Off := TRUE;
	Real_to_Word_Pos_Calib(	R_RB_X	:= TO_REAL(GVL.RB_B_.CUR_X),
				R_RB_Y	:= TO_REAL(GVL.RB_B_.CUR_Y),
				R_RB_r	:= TO_REAL(GVL.RB_B_.CUR_R),
				LOW_RB_X	=> GVL.MODBUS[i_Vs_Align*6 + 16],
				HIGH_RB_X	=> GVL.MODBUS[i_Vs_Align*6 + 17],
				LOW_RB_Y	=> GVL.MODBUS[i_Vs_Align*6 + 18],
				HIGH_RB_Y	=> GVL.MODBUS[i_Vs_Align*6 + 19],
				LOW_RB_R	=> GVL.MODBUS[i_Vs_Align*6 + 20],
				HIGH_RB_R	=> GVL.MODBUS[i_Vs_Align*6 + 21]);
	IF (i_Vs_Align = 11) THEN
		GVL.Pro4_.Man.Run_Calib_Pos_Done := TRUE;
	END_IF;			 
END_IF;
IF (T_Delay_Trigger_Calib.Q AND Trigger_Calib_Done.Q AND Run_One_Pos_Calib) THEN
	T_Delay_Trigger_Calib.IN := FALSE;
	GVL.Pro4_.Man.Trigger_Vs_Align_On_Off := FALSE;
	i_Vs_Align := i_Vs_Align + 1;
	Run_One_Pos_Calib := FALSE;
END_IF
	
//END_WHILE
END_ACTION

ACTION Robot_Calib_Vision:
//Run_Calib_VS_RB_A - CAM 1
IF GVL.Data_Calib_RB[1].Use THEN
	GVL.Auto_VS_RB[1].RTrig_Trigger_VS_Done(CLK := GVL.Auto_VS_RB[1].Trigger_Done);
	GVL.Auto_VS_RB[1].RTrig_Trigger_Calib_VS_Done(CLK := GVL.Auto_VS_RB[1].Calib_VS_Done);
	Run_Calib_VS_RB[1](Enable := GVL.g_aVisionConfig[1].Enable,
					  Start := GVL.Calib_Cam_RB[1].Start,
					  Reset := GVL.Calib_Cam_RB[1].Reset,
					  CameraID := GVL.g_aVisionConfig[1].CameraID,
					  Hand_No := GVL.g_aVisionConfig[1].Robot,
					  PointNo1 := (GVL.Data_Calib_RB[1].PointNo1),
					  Nb_Point_X := GVL.Data_Calib_RB[1].Nb_Point_X,
					  Nb_Point_Y := GVL.Data_Calib_RB[1].Nb_Point_Y,
					  Delta_X := GVL.Data_Calib_RB[1].Delta_X,
					  Delta_Y := GVL.Data_Calib_RB[1].Delta_Y,
					  Delta_A := GVL.Data_Calib_RB[1].Delta_A,
					  A_Error := Move_Point_Para_A.A_Error,
					  B_Error := Move_Point_Para_B.B_Error,
					  T_Delay_Trigger_time := GVL.Data_Calib_RB[1].Delay_Trigger_Time,
					  Run_Mode := GVL.Data_Calib_RB[1].Run_By_Array_Point,
					  Run_No_Trigger := GVL.Data_Calib_RB[1].Run_No_Trigger,
					  CurrentPoint_Run_A := Pos_run_manual_A,  // Toa do diem chay calib RB A
					  CurrentPoint_Run_B := Pos_run_manual_B,  // Toa do diem chay calib RB B
					  ARunP := run_calib_P_Cam_A, // Bien cho robot A chay PTP
					  BRunP := run_calib_P_Cam_B, // Bien cho robot B chay PTP
					  A_Comp    := A_Comp_Man, // Bien bao robot A da chay den diem muc tieu
					  B_Comp    := B_Comp_Man, // Bien bao robot B da chay den diem muc tieu
					  Trigger_RB := GVL.Auto_VS_RB[1].Trigger_VS, // Bien trigger robot A gui Vision
					  Triger_RB_Done := GVL.Auto_VS_RB[1].Trigger_Done, //Bien trigger done Vision gui robot A
					  Run_Calib_Pos_Done := GVL.Auto_VS_RB[1].Run_Pos_Calib_Done, // Bien bao da chay xong cac diem calib
					  Calib_Done := GVL.Auto_VS_RB[1].Calib_VS_Done,
					  );
	IF GVL.Man_Calib_RB[1].Run_Calib_VS THEN
		GVL.Calib_Cam_RB[1].Enable := TRUE;
		GVL.Calib_Cam_RB[1].Start := TRUE;
	ELSE
		GVL.Calib_Cam_RB[1].Enable := FALSE;
		GVL.Calib_Cam_RB[1].Start := FALSE;
	END_IF;
	
	IF Run_Calib_VS_RB[1].DoneAll THEN
		GVL.Man_Calib_RB[1].Run_Calib_VS := FALSE;
	END_IF
	//IF GVL.Man_Calib_RB[0].Calib_VS_Done THEN 
	IF GVL.Auto_VS_RB[1].RTrig_Trigger_Calib_VS_Done.Q THEN
		GVL.Calib_Cam_RB[1].Enable := FALSE;
		GVL.Calib_Cam_RB[1].Start := FALSE;
	END_IF
END_IF;
END_ACTION

METHOD M_CACULATOR_Z : BOOL
VAR_INPUT
	DATA, ID , Z_COUNT : WORD; // 0 : RBA --- 1 : RBB
	PITCH_Z : REAL;
	Up_Down : BOOL;
END_VAR
CASE DATA OF
	0:
		IF  Up_Down THEN
			Pos_run_auto_A.c.Z := GVL_1.DATA_RB_A.Z_POS[ID] - Z_COUNT* PITCH_Z ;
		ELSE
			Pos_run_auto_A.c.Z := GVL_1.DATA_RB_A.Z_POS[ID] + Z_COUNT* PITCH_Z ;
		END_IF;

	1:
		IF  Up_Down THEN
		Pos_run_auto_B.c.Z := GVL_1.DATA_RB_B.Z_POS[ID] - Z_COUNT* PITCH_Z ;
		ELSE
		Pos_run_auto_B.c.Z := GVL_1.DATA_RB_B.Z_POS[ID] + Z_COUNT* PITCH_Z ;	
		END_IF;
END_CASE;
END_METHOD

METHOD M_CHOOSE_POS : BOOL
VAR_INPUT
	DATA, ID : WORD; // 0 : RBA --- 1 : RBB
	XYR_CONST, Z_CONST : BOOL;
	
END_VAR
CASE DATA OF
	0:
		IF XYR_CONST  AND NOT Z_CONST THEN
			Pos_run_auto_A.c.X := POU_MONITOR_ROBOT.RB1_POS.c.X ;
			Pos_run_auto_A.c.Y := POU_MONITOR_ROBOT.RB1_POS.c.Y ;
			Pos_run_auto_A.c.Z := GVL_1.DATA_RB_A.Z_POS[ID] ;
			Pos_run_auto_A.c.A := POU_MONITOR_ROBOT.RB1_POS.c.A ;
		ELSIF NOT XYR_CONST AND Z_CONST THEN
			Pos_run_auto_A.c.X := GVL_1.DATA_RB_A.X_POS[ID];
			Pos_run_auto_A.c.Y := GVL_1.DATA_RB_A.Y_POS[ID];
			Pos_run_auto_A.c.Z := POU_MONITOR_ROBOT.RB1_POS.c.Z;
			Pos_run_auto_A.c.A := GVL_1.DATA_RB_A.R_POS[ID] ;
		ELSE
			Pos_run_auto_A.c.X := GVL_1.DATA_RB_A.X_POS[ID];
			Pos_run_auto_A.c.Y := GVL_1.DATA_RB_A.Y_POS[ID];
			Pos_run_auto_A.c.Z := GVL_1.DATA_RB_A.Z_POS[ID];
			Pos_run_auto_A.c.A := GVL_1.DATA_RB_A.R_POS[ID];				
		END_IF
	1:
		IF XYR_CONST  AND NOT Z_CONST THEN
			Pos_run_auto_B.c.X := POU_MONITOR_ROBOT.RB2_POS.c.X ;
			Pos_run_auto_B.c.Y := POU_MONITOR_ROBOT.RB2_POS.c.Y ;
			Pos_run_auto_B.c.Z := GVL_1.DATA_RB_B.Z_POS[ID] ;
			Pos_run_auto_B.c.A := POU_MONITOR_ROBOT.RB2_POS.c.A ;
		ELSIF NOT XYR_CONST AND Z_CONST THEN
			Pos_run_auto_B.c.X := GVL_1.DATA_RB_B.X_POS[ID];
			Pos_run_auto_B.c.Y := GVL_1.DATA_RB_B.Y_POS[ID];
			Pos_run_auto_B.c.Z := POU_MONITOR_ROBOT.RB2_POS.c.Z;
			Pos_run_auto_B.c.A := GVL_1.DATA_RB_B.R_POS[ID] ;
		ELSE
			Pos_run_auto_B.c.X := GVL_1.DATA_RB_B.X_POS[ID];
			Pos_run_auto_B.c.Y := GVL_1.DATA_RB_B.Y_POS[ID];
			Pos_run_auto_B.c.Z := GVL_1.DATA_RB_B.Z_POS[ID];
			Pos_run_auto_B.c.A := GVL_1.DATA_RB_B.R_POS[ID];				
		END_IF	
END_CASE
END_METHOD

METHOD M_CHOOSE_POS_Calib : BOOL
VAR_INPUT
	DATA, ID : WORD; // 0 : RBA --- 1 : RBB
	XYR_CONST, Z_CONST : BOOL;
	
END_VAR
CASE DATA OF
	0:
		Pos_run_manual_A.c.X := GVL_1.DATA_RB_A.X_POS[ID];
		Pos_run_manual_A.c.Y := GVL_1.DATA_RB_A.Y_POS[ID];
		Pos_run_manual_A.c.Z := GVL_1.DATA_RB_A.Z_POS[ID];
		Pos_run_manual_A.c.A := GVL_1.DATA_RB_A.R_POS[ID];				
	1:	
		Pos_run_manual_B.c.X := GVL_1.DATA_RB_B.X_POS[ID];
		Pos_run_manual_B.c.Y := GVL_1.DATA_RB_B.Y_POS[ID];
		Pos_run_manual_B.c.Z := GVL_1.DATA_RB_B.Z_POS[ID];
		Pos_run_manual_B.c.A := GVL_1.DATA_RB_B.R_POS[ID];					
END_CASE
END_METHOD

METHOD M_CHOOSE_POS_Man : BOOL
VAR_INPUT
	DATA, ID : WORD; // 0 : RBA --- 1 : RBB
	XYR_CONST, Z_CONST : BOOL;
	
END_VAR
CASE DATA OF
	0:
		IF XYR_CONST  AND NOT Z_CONST THEN
			Pos_run_manual_A.c.X := POU_MONITOR_ROBOT.RB1_POS.c.X ;
			Pos_run_manual_A.c.Y := POU_MONITOR_ROBOT.RB1_POS.c.Y ;
			Pos_run_manual_A.c.Z := GVL_1.DATA_RB_A.Z_POS[ID] ;
			Pos_run_manual_A.c.A := POU_MONITOR_ROBOT.RB1_POS.c.A ;
		ELSIF NOT XYR_CONST AND Z_CONST THEN
			Pos_run_manual_A.c.X := GVL_1.DATA_RB_A.X_POS[ID];
			Pos_run_manual_A.c.Y := GVL_1.DATA_RB_A.Y_POS[ID];
			Pos_run_manual_A.c.Z := POU_MONITOR_ROBOT.RB1_POS.c.Z;
			Pos_run_manual_A.c.A := GVL_1.DATA_RB_A.R_POS[ID] ;
		ELSE
			Pos_run_manual_A.c.X := GVL_1.DATA_RB_A.X_POS[ID];
			Pos_run_manual_A.c.Y := GVL_1.DATA_RB_A.Y_POS[ID];
			Pos_run_manual_A.c.Z := GVL_1.DATA_RB_A.Z_POS[ID];
			Pos_run_manual_A.c.A := GVL_1.DATA_RB_A.R_POS[ID];				
		END_IF
	1:
		IF XYR_CONST  AND NOT Z_CONST THEN
			Pos_run_manual_B.c.X := POU_MONITOR_ROBOT.RB2_POS.c.X ;
			Pos_run_manual_B.c.Y := POU_MONITOR_ROBOT.RB2_POS.c.Y ;
			Pos_run_manual_B.c.Z := GVL_1.DATA_RB_B.Z_POS[ID] ;
			Pos_run_manual_B.c.A := POU_MONITOR_ROBOT.RB2_POS.c.A ;
		ELSIF NOT XYR_CONST AND Z_CONST THEN
			Pos_run_manual_B.c.X := GVL_1.DATA_RB_B.X_POS[ID];
			Pos_run_manual_B.c.Y := GVL_1.DATA_RB_B.Y_POS[ID];
			Pos_run_manual_B.c.Z := POU_MONITOR_ROBOT.RB2_POS.c.Z;
			Pos_run_manual_B.c.A := GVL_1.DATA_RB_B.R_POS[ID] ;
		ELSE
			Pos_run_manual_B.c.X := GVL_1.DATA_RB_B.X_POS[ID];
			Pos_run_manual_B.c.Y := GVL_1.DATA_RB_B.Y_POS[ID];
			Pos_run_manual_B.c.Z := GVL_1.DATA_RB_B.Z_POS[ID];
			Pos_run_manual_B.c.A := GVL_1.DATA_RB_B.R_POS[ID];				
		END_IF	
END_CASE
END_METHOD

METHOD M_CHOOSE_POS_VS : BOOL
VAR_INPUT
	DATA, ID : WORD; // 0 : RBA --- 1 : RBB
	XYR_CONST, Z_CONST : BOOL;
	
END_VAR
CASE DATA OF
	0:
		IF NOT XYR_CONST AND Z_CONST THEN
			Pos_run_auto_A.c.X := GVL_1.DATA_RB_A.X_POS[ID] + GVL.Cam_T1.POS_X_OFFSET;
			Pos_run_auto_A.c.Y := GVL_1.DATA_RB_A.Y_POS[ID] + GVL.Cam_T1.POS_Y_OFFSET;
			Pos_run_auto_A.c.Z := POU_MONITOR_ROBOT.RB1_POS.c.Z;
			Pos_run_auto_A.c.A := GVL_1.DATA_RB_A.R_POS[ID] + GVL.Cam_T1.POS_R_OFFSET;			
		END_IF
	1:
		IF NOT XYR_CONST AND Z_CONST THEN
			Pos_run_auto_B.c.X := GVL_1.DATA_RB_B.X_POS[ID] + GVL.Cam_T1.POS_X_OFFSET;
			Pos_run_auto_B.c.Y := GVL_1.DATA_RB_B.Y_POS[ID] + GVL.Cam_T1.POS_Y_OFFSET;
			Pos_run_auto_B.c.Z := POU_MONITOR_ROBOT.RB2_POS.c.Z;
			Pos_run_auto_B.c.A := GVL_1.DATA_RB_B.R_POS[ID] + GVL.Cam_T1.POS_R_OFFSET;			
		END_IF	
END_CASE
END_METHOD

METHOD M_CHOOSE_POS_XY : BOOL
VAR_INPUT
	DATA, ID : WORD; // 0 : RBA --- 1 : RBB
	XY_CONST : BOOL;
	
END_VAR
CASE DATA OF
	0:
		IF XY_CONST THEN
			Pos_run_auto_A.c.X := GVL_1.DATA_RB_A.X_POS[ID] ;
			Pos_run_auto_A.c.Y := GVL_1.DATA_RB_A.Y_POS[ID] ;
			Pos_run_auto_A.c.Z := POU_MONITOR_ROBOT.RB1_POS.c.Z ;
			Pos_run_auto_A.c.A := POU_MONITOR_ROBOT.RB1_POS.c.A ;
		ELSE
			Pos_run_auto_A.c.X := GVL_1.DATA_RB_A.X_POS[ID];
			Pos_run_auto_A.c.Y := GVL_1.DATA_RB_A.Y_POS[ID];
			Pos_run_auto_A.c.Z := GVL_1.DATA_RB_A.Z_POS[ID];
			Pos_run_auto_A.c.A := GVL_1.DATA_RB_A.R_POS[ID];				
		END_IF
	1:
		IF XY_CONST  THEN
			Pos_run_auto_B.c.X := GVL_1.DATA_RB_B.X_POS[ID] ;
			Pos_run_auto_B.c.Y := GVL_1.DATA_RB_B.Y_POS[ID] ;
			Pos_run_auto_B.c.Z := POU_MONITOR_ROBOT.RB2_POS.c.Z ;
			Pos_run_auto_B.c.A := POU_MONITOR_ROBOT.RB2_POS.c.A ;
		ELSE
			Pos_run_auto_B.c.X := GVL_1.DATA_RB_B.X_POS[ID];
			Pos_run_auto_B.c.Y := GVL_1.DATA_RB_B.Y_POS[ID];
			Pos_run_auto_B.c.Z := GVL_1.DATA_RB_B.Z_POS[ID];
			Pos_run_auto_B.c.A := GVL_1.DATA_RB_B.R_POS[ID];				
		END_IF	
END_CASE
END_METHOD

METHOD M_CHOOSE_POS_Z_BF : BOOL
VAR_INPUT
	DATA, ID : WORD; // 0 : RBA --- 1 : RBB
	XYR_CONST, Z_CONST : BOOL;
	
END_VAR
CASE DATA OF
	0:
		IF XYR_CONST  AND NOT Z_CONST THEN
			Pos_run_auto_A.c.X := POU_MONITOR_ROBOT.RB1_POS.c.X ;
			Pos_run_auto_A.c.Y := POU_MONITOR_ROBOT.RB1_POS.c.Y ;
			Pos_run_auto_A.c.Z := GVL_1.DATA_RB_A.Z_POS[ID] + 10 ;
			Pos_run_auto_A.c.A := POU_MONITOR_ROBOT.RB1_POS.c.A ;
		ELSIF NOT XYR_CONST AND Z_CONST THEN
			Pos_run_auto_A.c.X := GVL_1.DATA_RB_A.X_POS[ID];
			Pos_run_auto_A.c.Y := GVL_1.DATA_RB_A.Y_POS[ID];
			Pos_run_auto_A.c.Z := POU_MONITOR_ROBOT.RB1_POS.c.Z;
			Pos_run_auto_A.c.A := GVL_1.DATA_RB_A.R_POS[ID] ;
		ELSE
			Pos_run_auto_A.c.X := GVL_1.DATA_RB_A.X_POS[ID];
			Pos_run_auto_A.c.Y := GVL_1.DATA_RB_A.Y_POS[ID];
			Pos_run_auto_A.c.Z := GVL_1.DATA_RB_A.Z_POS[ID] + 10;
			Pos_run_auto_A.c.A := GVL_1.DATA_RB_A.R_POS[ID];				
		END_IF
	1:
		IF XYR_CONST  AND NOT Z_CONST THEN
			Pos_run_auto_B.c.X := POU_MONITOR_ROBOT.RB2_POS.c.X ;
			Pos_run_auto_B.c.Y := POU_MONITOR_ROBOT.RB2_POS.c.Y ;
			Pos_run_auto_B.c.Z := GVL_1.DATA_RB_B.Z_POS[ID] + 10 ;
			Pos_run_auto_B.c.A := POU_MONITOR_ROBOT.RB2_POS.c.A ;
		ELSIF NOT XYR_CONST AND Z_CONST THEN
			Pos_run_auto_B.c.X := GVL_1.DATA_RB_B.X_POS[ID];
			Pos_run_auto_B.c.Y := GVL_1.DATA_RB_B.Y_POS[ID];
			Pos_run_auto_B.c.Z := POU_MONITOR_ROBOT.RB2_POS.c.Z;
			Pos_run_auto_B.c.A := GVL_1.DATA_RB_B.R_POS[ID] ;
		ELSE
			Pos_run_auto_B.c.X := GVL_1.DATA_RB_B.X_POS[ID];
			Pos_run_auto_B.c.Y := GVL_1.DATA_RB_B.Y_POS[ID];
			Pos_run_auto_B.c.Z := GVL_1.DATA_RB_B.Z_POS[ID] + 10;
			Pos_run_auto_B.c.A := GVL_1.DATA_RB_B.R_POS[ID];				
		END_IF	
END_CASE
END_METHOD

METHOD M_initProcess
IF GVL.MB_[6] AND GVL.RB_A.Manual AND GVL.RB_B.Manual THEN
	GVL_2.Project2_RB_A_Get.P1_Z_ :=  GVL_2.Project2_RB_A_Get.P1_Z;	 
	GVL_2.Project2_RB_A_Get.P2_Z_ :=  GVL_2.Project2_RB_A_Get.P2_Z;	
	GVL_2.Project2_RB_A_Get.P3_Z_ :=  GVL_2.Project2_RB_A_Get.P3_Z;  
	GVL_2.Project2_RB_A_Get.P4_Z_ :=  GVL_2.Project2_RB_A_Get.P4_Z;
	
	GVL_2.Project2_RB_A_Put.P1_Z_ :=  0;	 
	GVL_2.Project2_RB_A_Put.P2_Z_ :=  0;
	GVL_2.Project2_RB_A_Put.P3_Z_ :=  0;  
	GVL_2.Project2_RB_A_Put.P4_Z_ :=  0;
	
	GVL_2.Project2_RB_B_Get.P1_Z_ := 0;
	GVL_2.Project2_RB_B_Get.P2_Z_ := 0;
	GVL_2.Project2_RB_B_Get.P3_Z_ := 0;
	GVL_2.Project2_RB_B_Get.P4_Z_ := 0;

	GVL_2.Project2_RB_B_Put.P1_Z_ := 0;
	GVL_2.Project2_RB_B_Put.P2_Z_ := 0;
	GVL_2.Project2_RB_B_Put.P3_Z_ := 0;
	GVL_2.Project2_RB_B_Put.P4_Z_ := 0;	
	
	GVL.RB_A_.Tool_1 := FALSE;
	GVL.RB_B_.Tool_1 := FALSE;
END_IF;	

IF GVL.MB_[7] AND GVL.RB_A.Manual AND GVL.RB_B.Manual THEN
	GVL_2.Project2_RB_B_Get.P1_Z_ :=  GVL_2.Project2_RB_B_Get.P1_Z;	 
	GVL_2.Project2_RB_B_Get.P2_Z_ :=  GVL_2.Project2_RB_B_Get.P2_Z;	
	GVL_2.Project2_RB_B_Get.P3_Z_ :=  GVL_2.Project2_RB_B_Get.P3_Z;  
	GVL_2.Project2_RB_B_Get.P4_Z_ :=  GVL_2.Project2_RB_B_Get.P4_Z;
	
	GVL_2.Project2_RB_B_Put.P1_Z_ :=  0;	 
	GVL_2.Project2_RB_B_Put.P2_Z_ :=  0;
	GVL_2.Project2_RB_B_Put.P3_Z_ :=  0;  
	GVL_2.Project2_RB_B_Put.P4_Z_ :=  0;
	
	GVL.RB_A_.Tool_1 := FALSE;
	GVL.RB_B_.Tool_1 := FALSE;
END_IF;
END_METHOD

METHOD M_R_Mov : Bool
VAR_INPUT
	DATA, ID : WORD; // 0 : RBA --- 1 : RBB
	R_,Z_,X_,Y_ : BOOL;
END_VAR
CASE DATA OF
	0:
		IF R_ AND NOT X_ AND NOT Y_ AND NOT Z_ THEN
			Pos_run_auto_A.c.X := POU_MONITOR_ROBOT.RB1_POS.c.X ;
			Pos_run_auto_A.c.Y := POU_MONITOR_ROBOT.RB1_POS.c.Y ;
			Pos_run_auto_A.c.Z := POU_MONITOR_ROBOT.RB1_POS.c.Z ;
			Pos_run_auto_A.c.A := GVL_1.DATA_RB_A.R_POS[ID] ;
		ELSIF NOT R_ AND X_ AND NOT Y_ AND NOT Z_ THEN
			Pos_run_auto_A.c.X := GVL_1.DATA_RB_A.X_POS[ID] ;
			Pos_run_auto_A.c.Y := POU_MONITOR_ROBOT.RB1_POS.c.Y ;
			Pos_run_auto_A.c.Z := POU_MONITOR_ROBOT.RB1_POS.c.Z ;
			Pos_run_auto_A.c.A := POU_MONITOR_ROBOT.RB1_POS.c.A ;
		ELSIF NOT R_ AND NOT X_ AND  Y_ AND NOT Z_ THEN
			Pos_run_auto_A.c.X := POU_MONITOR_ROBOT.RB1_POS.c.X ;
			Pos_run_auto_A.c.Y := GVL_1.DATA_RB_A.Y_POS[ID] ;
			Pos_run_auto_A.c.Z := POU_MONITOR_ROBOT.RB1_POS.c.Z ;
			Pos_run_auto_A.c.A := POU_MONITOR_ROBOT.RB1_POS.c.A ;	
		ELSIF NOT R_ AND NOT X_ AND NOT Y_ AND Z_ THEN
			Pos_run_auto_A.c.X := POU_MONITOR_ROBOT.RB1_POS.c.X ;
			Pos_run_auto_A.c.Y := POU_MONITOR_ROBOT.RB1_POS.c.Y ;
			Pos_run_auto_A.c.Z := GVL_1.DATA_RB_A.Z_POS[ID] ;
			Pos_run_auto_A.c.A := POU_MONITOR_ROBOT.RB1_POS.c.A ;			
		ELSIF NOT R_ AND  X_ AND Y_ AND NOT Z_ THEN
			Pos_run_auto_A.c.X := GVL_1.DATA_RB_A.X_POS[ID] ;
			Pos_run_auto_A.c.Y := GVL_1.DATA_RB_A.Y_POS[ID] ;
			Pos_run_auto_A.c.Z := POU_MONITOR_ROBOT.RB1_POS.c.Z ;
			Pos_run_auto_A.c.A := POU_MONITOR_ROBOT.RB1_POS.c.A ;				
		END_IF
	1:
		IF R_ AND NOT X_ AND NOT Y_ AND NOT Z_ THEN
			Pos_run_auto_B.c.X := POU_MONITOR_ROBOT.RB2_POS.c.X ;
			Pos_run_auto_B.c.Y := POU_MONITOR_ROBOT.RB2_POS.c.Y ;
			Pos_run_auto_B.c.Z := POU_MONITOR_ROBOT.RB2_POS.c.Z ;
			Pos_run_auto_B.c.A := GVL_1.DATA_RB_B.R_POS[ID] ;
		ELSIF NOT R_ AND X_ AND NOT Y_ AND NOT Z_ THEN
			Pos_run_auto_B.c.X := GVL_1.DATA_RB_B.X_POS[ID] ;
			Pos_run_auto_B.c.Y := POU_MONITOR_ROBOT.RB2_POS.c.Y ;
			Pos_run_auto_B.c.Z := POU_MONITOR_ROBOT.RB2_POS.c.Z ;
			Pos_run_auto_B.c.A := POU_MONITOR_ROBOT.RB2_POS.c.A ;
		ELSIF NOT R_ AND NOT X_ AND  Y_ AND NOT Z_ THEN
			Pos_run_auto_B.c.X := POU_MONITOR_ROBOT.RB2_POS.c.X ;
			Pos_run_auto_B.c.Y := GVL_1.DATA_RB_B.Y_POS[ID] ;
			Pos_run_auto_B.c.Z := POU_MONITOR_ROBOT.RB2_POS.c.Z ;
			Pos_run_auto_B.c.A := POU_MONITOR_ROBOT.RB2_POS.c.A ;	
		ELSIF NOT R_ AND NOT X_ AND NOT Y_ AND Z_ THEN
			Pos_run_auto_B.c.X := POU_MONITOR_ROBOT.RB2_POS.c.X ;
			Pos_run_auto_B.c.Y := POU_MONITOR_ROBOT.RB2_POS.c.Y ;
			Pos_run_auto_B.c.Z := GVL_1.DATA_RB_B.Z_POS[ID] ;
			Pos_run_auto_B.c.A := POU_MONITOR_ROBOT.RB2_POS.c.A ;	
		ELSIF NOT R_ AND  X_ AND Y_ AND NOT Z_ THEN
			Pos_run_auto_B.c.X := GVL_1.DATA_RB_B.X_POS[ID] ;
			Pos_run_auto_B.c.Y := GVL_1.DATA_RB_B.Y_POS[ID] ;
			Pos_run_auto_B.c.Z := POU_MONITOR_ROBOT.RB2_POS.c.Z ;
			Pos_run_auto_B.c.A := POU_MONITOR_ROBOT.RB2_POS.c.A ;				
		END_IF
END_CASE
END_METHOD

METHOD M_reset
IF NOT GVL.X[9] THEN // EMG

Excute_Run_goHome_a := FALSE;
AP_Man_Z_Wait_Go := FALSE;
AP_Man_R_Wait_Go := FALSE;
AP_Man_XY_Wait_Go := FALSE;
AP_Man_Pos_Go := FALSE;
AP_Man_Pos_Go_L := FALSE;
AP_Man_UP_Z_Go := FALSE;
//excute_run_P_cam_a := FALSE;
//run_P_cam_a_test_pick := FALSE;
//run_P_cam_a_test_place := FALSE;
AP_Auto_Pos_Go  := FALSE;

A3_Run_P := FALSE; A3_Run_L := FALSE;

Excute_Run_goHome_B := FALSE; Excute_Run_goZ_Wait_B := FALSE; Excute_Run_goR_Wait_B := FALSE; Excute_Run_goXY_Wait_B := FALSE;



Excute_Run_goPos_B := FALSE; excute_run_P_Upz_B := FALSE; Excute_Run_goPos_B_L := FALSE;

excute_run_P_cam_B := FALSE; run_P_cam_B_test_pick := FALSE; run_P_cam_B_test_place := FALSE;



EXCUTE_RUN_P_AUTO_B  := FALSE;

Running_B_Cam := FALSE;

B3_Run_P := FALSE; B3_Run_L := FALSE;	
END_IF
END_METHOD

ACTION ACT_Excute_Run:
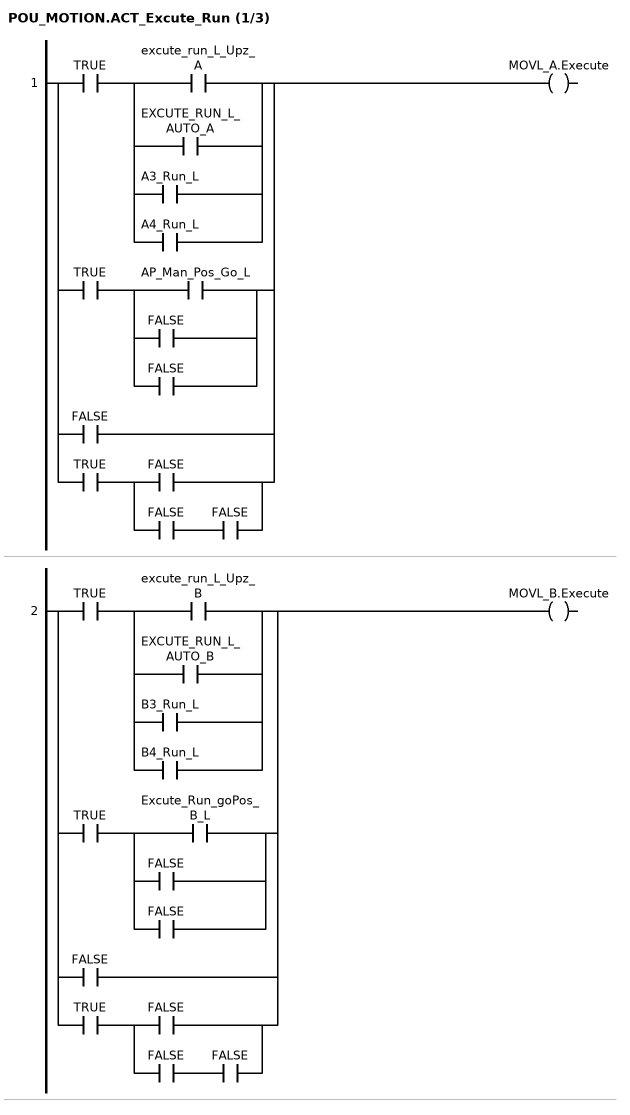
// NETWORK 1
MOVL_A.Execute := (TRUE AND excute_run_L_Upz_A OR TRUE AND EXCUTE_RUN_L_AUTO_A OR TRUE AND A3_Run_L OR TRUE AND A4_Run_L) OR (TRUE AND AP_Man_Pos_Go_L OR TRUE AND FALSE OR TRUE AND FALSE) OR FALSE OR (TRUE AND FALSE OR (TRUE AND FALSE) AND FALSE);

// NETWORK 2
MOVL_B.Execute := (TRUE AND excute_run_L_Upz_B OR TRUE AND EXCUTE_RUN_L_AUTO_B OR TRUE AND B3_Run_L OR TRUE AND B4_Run_L) OR (TRUE AND Excute_Run_goPos_B_L OR TRUE AND FALSE OR TRUE AND FALSE) OR FALSE OR (TRUE AND FALSE OR (TRUE AND FALSE) AND FALSE);

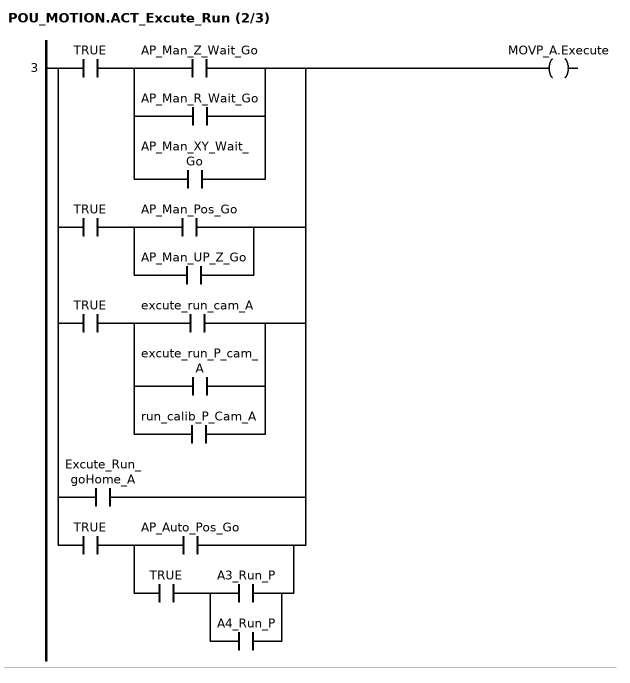
// NETWORK 3
MOVP_A.Execute := (TRUE AND AP_Man_Z_Wait_Go OR TRUE AND AP_Man_R_Wait_Go OR TRUE AND AP_Man_XY_Wait_Go) OR (TRUE AND AP_Man_Pos_Go OR TRUE AND AP_Man_UP_Z_Go) OR TRUE AND (excute_run_cam_A OR excute_run_P_cam_A OR run_calib_P_Cam_A) OR Excute_Run_goHome_A OR (TRUE AND AP_Auto_Pos_Go OR (TRUE AND TRUE) AND (A3_Run_P OR A4_Run_P));

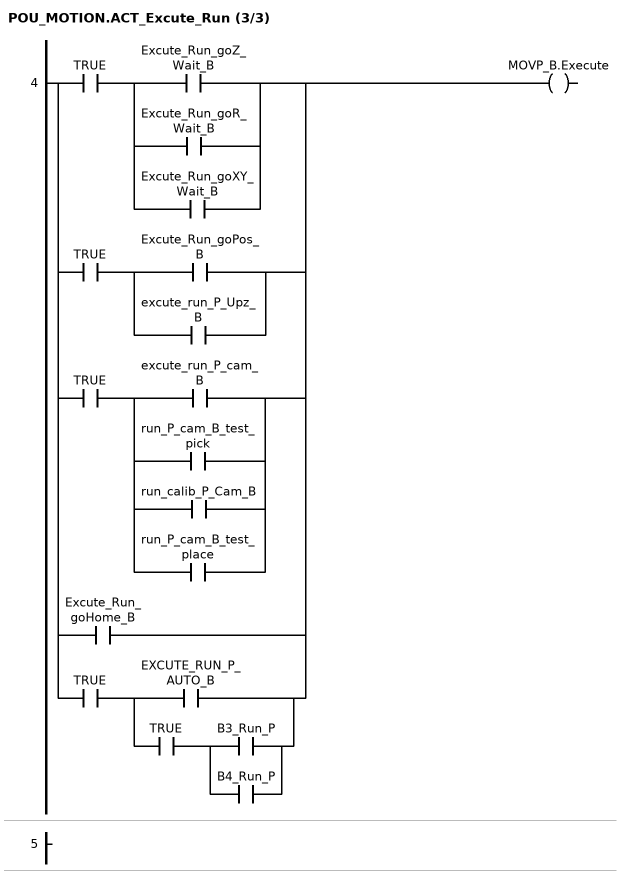
// NETWORK 4
MOVP_B.Execute := (TRUE AND Excute_Run_goZ_Wait_B OR TRUE AND Excute_Run_goR_Wait_B OR TRUE AND Excute_Run_goXY_Wait_B) OR (TRUE AND Excute_Run_goPos_B OR TRUE AND excute_run_P_Upz_B) OR TRUE AND (excute_run_P_cam_B OR run_P_cam_B_test_pick OR run_calib_P_Cam_B OR run_P_cam_B_test_place) OR Excute_Run_goHome_B OR (TRUE AND EXCUTE_RUN_P_AUTO_B OR (TRUE AND TRUE) AND (B3_Run_P OR B4_Run_P));

// NETWORK 5
END_ACTION

END_PROGRAM

// Just_Motion_Control_x86_64_Linux_SM_WV/Application/FB_/FB_Write_Log
FUNCTION_BLOCK FB_Write_Log
VAR_OUTPUT
    Logs : ARRAY[0..20] OF STRING[255];
END_VAR

VAR
    Buffer : ARRAY[0..20] OF STRING[255];
    Index : INT := 1;

    tMs : UDINT;
	
	Hour   : UDINT;
    Minute : UDINT;
    Second : UDINT;
	
    TimeStr : STRING[30];
    TempStr : STRING[255];

    i : INT;
	Logs_old : STRING[255];
END_VAR

(* sắp xếp log mới nhất lên trên *)
// FOR i := 1 TO 20 DO
// 
//     IF (Index - i) > 0 THEN
//         Logs[i] := Buffer[Index - i];
//     ELSE
//         Logs[i] := Buffer[20 + (Index - i)];
//     END_IF
// 
// END_FOR

METHOD Write
VAR_INPUT
    Message : STRING[255];
END_VAR
VAR
    LastMessage : STRING[255];
	 dt_          : DWORD;
END_VAR
(* nếu message giống lần trước thì bỏ qua *)
IF Message = Logs_old THEN
    RETURN;
ELSIF Message <> Logs_old THEN

//tMs := SysTimeGetMs();
(* Lấy thời gian thực *)
//SysTimeRtcGet(pResult := 7,SysTimeRtcGet => dt_ );

(* Quy đổi *)
// Hour := tMs / 3600000;
// Minute := (tMs / 60000) MOD 60;
// Second := (tMs / 1000) MOD 60;

Second := GVL.DW_[30];
Minute := GVL.DW_[31];
Hour := GVL.DW_[32];

(* Format hh:mm:ss *)
TimeStr := '';

(* Hour *)
IF Hour < 10 THEN
    TimeStr := CONCAT('0', UDINT_TO_STRING(Hour));
ELSE
    TimeStr := UDINT_TO_STRING(Hour);
END_IF

TimeStr := CONCAT(TimeStr, ':');

(* Minute *)
IF Minute < 10 THEN
    TimeStr := CONCAT(TimeStr, CONCAT('0', UDINT_TO_STRING(Minute)));
ELSE
    TimeStr := CONCAT(TimeStr, UDINT_TO_STRING(Minute));
END_IF

TimeStr := CONCAT(TimeStr, ':');

(* Second *)
IF Second < 10 THEN
    TimeStr := CONCAT(TimeStr, CONCAT('0', UDINT_TO_STRING(Second)));
ELSE
    TimeStr := CONCAT(TimeStr, UDINT_TO_STRING(Second));
END_IF

(* Ghép chuỗi *)
TempStr := CONCAT(TimeStr, ' | ');
TempStr := CONCAT(TempStr, Message);

Buffer[Index] := TempStr;

Logs_old := Message;

Index := Index + 1;

IF Index > 20 THEN
    Index := 1;
END_IF
LastMessage := Message;
END_IF;
END_METHOD

END_FUNCTION_BLOCK

// Just_Motion_Control_x86_64_Linux_SM_WV/Application/FB_/FB_PALLETS
FUNCTION_BLOCK FB_PALLETS
VAR_INPUT
    Enable      : BOOL;
    Inc         : BOOL;
    Dec         : BOOL;

    PalletMode  : INT; // 0:= PUT / 1 := GET
    ZOrder      : INT; //0:= Z trước hay 1:= Z sau
    RowFirst    : BOOL;// TRUE = Row trước, FALSE = Col trước

    RowCount    : INT;
    ColCount    : INT;
    ZCount      : INT;

    PitchRow    : REAL;
    PitchCol    : REAL;
    PitchZ      : REAL;

    StartX      : REAL;
    StartY      : REAL;
    StartZ      : REAL;
END_VAR
VAR_OUTPUT
    CurrentID   : INT;

    RowIndex    : INT;
    ColIndex    : INT;
    ZIndex      : INT;

    PosX        : REAL;
    PosY        : REAL;
    PosZ        : REAL;

    MaxID       : INT;
END_VAR
VAR
    IncTrig : R_TRIG;
    DecTrig : R_TRIG;
END_VAR

MaxID := RowCount * ColCount * ZCount;
{region "1. KHOI TAO PUT/GET"}
IF NOT Enable THEN
    CASE PalletMode OF
        0:
            CurrentID := 0;
        1:
            CurrentID := MaxID - 1;
    END_CASE;
END_IF;
{endregion}	 
{region "2. LOGIC INC/DEC ID"}
IncTrig(CLK := Inc);
DecTrig(CLK := Dec);

IF Enable THEN
    CASE PalletMode OF

        // ===== GET =====
        0:
            IF IncTrig.Q AND (CurrentID < MaxID - 1) THEN
                CurrentID := CurrentID + 1;
            END_IF;

            IF DecTrig.Q AND (CurrentID > 0) THEN
                CurrentID := CurrentID - 1;
            END_IF;

        // ===== PUT =====
        1:
            IF IncTrig.Q AND (CurrentID > 0) THEN
                CurrentID := CurrentID - 1;
            END_IF;

            IF DecTrig.Q AND (CurrentID < MaxID - 1) THEN
                CurrentID := CurrentID + 1;
            END_IF;

    END_CASE;
END_IF;
{endregion}	 
{region "3. LOGIC ROW/COLUMN/ZCOUNT"}	 
// Z TRƯỚC
IF ZOrder = 0 THEN

    ZIndex := CurrentID MOD ZCount;

    IF RowFirst AND  ZCount <> 0 THEN
        ColIndex := (CurrentID / ZCount) MOD ColCount;
        RowIndex := CurrentID / (ZCount * ColCount);
    ELSIF NOT  RowFirst AND ZCount <> 0 THEN
        RowIndex := (CurrentID / ZCount) MOD RowCount;
        ColIndex := CurrentID / (ZCount * RowCount);
    END_IF;

END_IF;
// Z SAU	 
IF ZOrder = 1 THEN

    ZIndex := CurrentID / (RowCount * ColCount);

    IF RowFirst AND ColCount <> 0 THEN
        RowIndex := (CurrentID MOD (RowCount * ColCount)) / ColCount;
        ColIndex := (CurrentID MOD (RowCount * ColCount)) MOD ColCount;
    ELSIF NOT RowFirst AND  ColCount <> 0 THEN
        ColIndex := (CurrentID MOD (RowCount * ColCount)) / RowCount;
        RowIndex := (CurrentID MOD (RowCount * ColCount)) MOD RowCount;
    END_IF;

END_IF;
{endregion}	 	 
{region "4. CACULATOR XYZ"}	 
PosX := StartX + ColIndex * PitchCol;
PosY := StartY + RowIndex * PitchRow;
PosZ := StartZ + ZIndex * PitchZ;
{endregion}

END_FUNCTION_BLOCK

// Just_Motion_Control_x86_64_Linux_SM_WV/Application/FB_/Blink_Bit
FUNCTION_BLOCK Blink_Bit
VAR_INPUT
	Enable     : BOOL;        // Cho phép blink
    TON_Time   : TIME := T#500ms; // Thời gian ON
    TOFF_Time  : TIME := T#500ms; // Thời gian OFF
END_VAR
VAR_OUTPUT
	 Out        : BOOL;        // Bit nhấp nháy
END_VAR
VAR
	ton        : TON;         // Timer ON
    toff       : TON;         // Timer OFF
    state      : BOOL := FALSE; // FALSE = OFF, TRUE = ON
END_VAR

IF NOT Enable THEN
    Out := FALSE;
    state := FALSE;
    ton(IN := FALSE);
    toff(IN := FALSE);
ELSE
    IF state = FALSE THEN
        ton(IN := TRUE, PT := TON_Time);

        IF ton.Q THEN
            ton(IN := FALSE);
            state := TRUE;
        END_IF

        Out := FALSE;

    ELSE
        toff(IN := TRUE, PT := TOFF_Time);

        IF toff.Q THEN
            toff(IN := FALSE);
            state := FALSE;
        END_IF

        Out := TRUE;
    END_IF
END_IF

END_FUNCTION_BLOCK

// Just_Motion_Control_x86_64_Linux_SM_WV/Application/FB_/FB_Run_Point
FUNCTION_BLOCK PUBLIC FB_Run_Point
VAR_INPUT
	Enable	  : BOOL;
	Hand_Type : INT; // 0: Trai-A; 1: Phai-B
	Move_Type : INT; // 0: MovP ; 1-MovL; 2-MovC
	A_Error   : BOOL;
	B_Error   : BOOL;
	A_Ready : BOOL;
	B_Ready : BOOL;
END_VAR
VAR_IN_OUT
	ARunP : BOOL;
    ARunL : BOOL;
	BRunP : BOOL;
    BRunL : BOOL;
	A_Comp    : BOOL;
	B_Comp    : BOOL;
END_VAR
VAR_OUTPUT
	Done : BOOL;  // Da chay xong target pos
	Busy : BOOL;  // Dang chay target pos
	Error : BOOL; // Function Error
END_VAR

IF NOT Enable THEN
	Error := FALSE;
	Done := FALSE; 	
	Busy := FALSE;
	IF Hand_Type = 0 THEN
		ARunP := FALSE;
		ARunL := FALSE;
	END_IF;
	IF Hand_Type = 1 THEN
		BRunP := FALSE;
		BRunL := FALSE;
	END_IF;
	RETURN;
END_IF

IF A_Error AND Hand_Type = 0  THEN
    Error := FALSE;
	Done := FALSE; 	
	Busy := FALSE;
	ARunP := FALSE;
	ARunL := FALSE;
	RETURN;
END_IF;

IF B_Error AND Hand_Type = 1  THEN
    Error := FALSE;
	Done := FALSE; 	
	Busy := FALSE;
	BRunP := FALSE;
	BRunL := FALSE;
	RETURN;
END_IF;

IF Enable THEN
	IF Hand_Type = 0 THEN  // Robot Trai - A
		IF Move_Type = 0 THEN // MovP
			IF NOT ARunP AND NOT A_Comp AND NOT Busy AND A_Ready AND NOT Done AND NOT Busy THEN
				A_Comp := FALSE;
				ARunP := TRUE;
				Busy := TRUE;
			END_IF						
			IF A_Comp AND ARunP THEN
				ARunP	 := FALSE;
				A_Comp	 := FALSE;
				Busy := FALSE;
				Done	 := TRUE;
			END_IF
		END_IF	
		IF Move_Type = 1 THEN // MovL
			IF NOT ARunL AND NOT A_Comp AND NOT Busy AND A_Ready AND NOT Done AND NOT Busy THEN
				A_Comp := FALSE;
				ARunL := TRUE;
				Busy := TRUE;
			END_IF						
			IF A_Comp AND ARunL THEN
				ARunL	 := FALSE;
				A_Comp	 := FALSE;
				Busy := FALSE;
				Done	 := TRUE;
			END_IF
		END_IF	
	END_IF
	// RB B
	IF Hand_Type = 1 THEN  // Robot Phai - B
		IF Move_Type = 0 THEN // MovP
			IF NOT BRunP AND NOT B_Comp AND NOT Busy AND B_Ready AND NOT Done AND NOT Busy THEN
				B_Comp := FALSE;
				BRunP := TRUE;
				Busy := TRUE;
			END_IF						
			IF B_Comp AND BRunP THEN
				BRunP	 := FALSE;
				B_Comp	 := FALSE;
				Busy := FALSE;
				Done	 := TRUE;
			END_IF
		END_IF	
		IF Move_Type = 1 THEN // MovL
			IF NOT BRunL AND NOT B_Comp AND NOT Busy AND B_Ready AND NOT Done AND NOT Busy THEN
				B_Comp := FALSE;
				BRunL := TRUE;
				Busy := TRUE;
			END_IF						
			IF B_Comp AND BRunL THEN
				BRunL	 := FALSE;
				B_Comp	 := FALSE;
				Busy := FALSE;
				Done	 := TRUE;
			END_IF
		END_IF	
	END_IF
END_IF

END_FUNCTION_BLOCK

// Just_Motion_Control_x86_64_Linux_SM_WV/Application/FB_/FB_Real_TO_Word_
FUNCTION_BLOCK FB_Real_TO_Word_
VAR_INPUT
	R_RB_X, R_RB_Y, R_RB_R : REAL;
END_VAR
VAR_OUTPUT
	HIGH_RB_X , LOW_RB_X,
	HIGH_RB_Y , LOW_RB_Y,
	HIGH_RB_R , LOW_RB_R : WORD;
END_VAR
	
VAR
	DINT_RB_X, DINT_RB_Y, DINT_RB_R : DINT;
	W_LOW_RB_X, W_HIGH_RB_X,
	W_LOW_RB_Y, W_HIGH_RB_Y,
	W_LOW_RB_R, W_HIGH_RB_R : WORD;
END_VAR

    DINT_RB_X := REAL_TO_DINT(R_RB_X*1000);
	DINT_RB_Y := REAL_TO_DINT(R_RB_Y*1000);
	DINT_RB_R := REAL_TO_DINT(R_RB_R*1000);

	W_HIGH_RB_X := DINT_TO_WORD(SHR(DINT_RB_X, 16));  // Lấy 16 bit cao
	W_LOW_RB_X := UDINT_TO_WORD(DINT_TO_UDINT( DINT_RB_X) AND 16#FFFF); // Lấy 16 bit thấp	
	W_HIGH_RB_Y := DINT_TO_WORD(SHR(DINT_RB_Y, 16));  // Lấy 16 bit cao
	W_LOW_RB_Y := UDINT_TO_WORD(DINT_TO_UDINT(DINT_RB_Y) AND 16#FFFF); // Lấy 16 bit thấp
	W_HIGH_RB_R := DINT_TO_WORD(SHR(DINT_RB_R, 16));  // Lấy 16 bit cao
	W_LOW_RB_R := UDINT_TO_WORD(DINT_TO_UDINT(DINT_RB_R) AND 16#FFFF); // Lấy 16 bit thấp
	
	LOW_RB_X:= W_LOW_RB_X;
	HIGH_RB_X := W_HIGH_RB_X;
	LOW_RB_Y := W_LOW_RB_Y;
	HIGH_RB_Y := W_HIGH_RB_Y;
	LOW_RB_R := W_LOW_RB_R;
	HIGH_RB_R := W_HIGH_RB_R;

END_FUNCTION_BLOCK

// Just_Motion_Control_x86_64_Linux_SM_WV/Application/FB_/FB_CalibRunPoints
FUNCTION_BLOCK FB_CalibRunPoints

VAR_INPUT
    Enable : BOOL;
    Start : BOOL;
    Reset : BOOL;

    CameraID : UINT; // Camera theo framework Vision moi: 1..GVL.C_MAX_VISION_CHANNELS

    Hand_No : INT;
    PointNo1 : INT; // So thu tu diem calib dau tien

    Nb_Point_X : INT;
    Nb_Point_Y : INT;

    Delta_X : INT; // Khoang cach giua cac diem theo phuong X
    Delta_Y : INT; // Khoang cach giua cac diem theo phuong Y
    Delta_A : INT; // Khoang cach giua cac diem theo phuong xoay

    A_Error : BOOL;
    B_Error : BOOL;

    T_Delay_Trigger_time : INT;

    Run_Mode : BOOL; // TRUE = sinh diem theo quy luat, FALSE = chay array diem day san
    Run_No_Trigger : BOOL; // TRUE = chi chay robot, khong giao tiep Vision
END_VAR


VAR_IN_OUT
    CurrentPoint_Run_A : SM3_Robotics.SMC_POS_REF; // Toa do diem chay calib Robot A
    CurrentPoint_Run_B : SM3_Robotics.SMC_POS_REF; // Toa do diem chay calib Robot B

    ARunP : BOOL; // Lenh PTP Robot A
    BRunP : BOOL; // Lenh PTP Robot B

    A_Comp : BOOL; // Robot A da den diem muc tieu
    B_Comp : BOOL; // Robot B da den diem muc tieu

    // Tam thoi GIU de khong vo interface cu.
    // Sau khi noi framework Vision moi on dinh se bo.
    Trigger_RB : BOOL;
    Triger_RB_Done : BOOL;
    Run_Calib_Pos_Done : BOOL;
    Calib_Done : BOOL;
END_VAR


VAR_OUTPUT
    Busy : BOOL;
    DoneAll : BOOL;
    Error : BOOL;
    ErrorID : INT;

    CurrentIndex : INT;
    PointCount : INT;
END_VAR


VAR
    State : INT;
    StartOld : BOOL;

    tTimeout : TON;
    t_Delay_Trigger : TON;

    Tmp_Delta : ST_POS;

    FTrig_Enable : F_TRIG;
    RTrig_Enable : R_TRIG;

    i_vs : INT;

    Trigger_Done_Old : BOOL;
    Calib_Done_Old : BOOL;
END_VAR

PointCount := Nb_Point_X * Nb_Point_Y;

t_Delay_Trigger(PT := TO_TIME(T_Delay_Trigger_time) * 100);

RTrig_Enable(CLK := Enable);

IF RTrig_Enable.Q THEN
    IF CameraID >= 1 AND CameraID <= GVL.C_MAX_VISION_CHANNELS THEN
        GVL.g_aVisionModbusControl[CameraID].RunCalib := FALSE;
        GVL.g_aVisionModbusControl[CameraID].CalibPosReady := FALSE;
        GVL.g_aVisionModbusControl[CameraID].CalibPointCount := 0;

        FOR i_vs := 1 TO 12 DO
            GVL.g_aVisionModbusControl[CameraID].CalibrationPoints[i_vs].X := 0.0;
            GVL.g_aVisionModbusControl[CameraID].CalibrationPoints[i_vs].Y := 0.0;
            GVL.g_aVisionModbusControl[CameraID].CalibrationPoints[i_vs].Z := 0.0;
            GVL.g_aVisionModbusControl[CameraID].CalibrationPoints[i_vs].A := 0.0;
        END_FOR;
    END_IF;
END_IF;
 
FTrig_Enable(CLK := Enable);
IF FTrig_Enable.Q THEN
	IF Hand_No = 1 THEN
		ARunP := FALSE;
	END_IF
	IF Hand_No = 2 THEN
		BRunP := FALSE;
	END_IF
	Trigger_RB := FALSE;
	Run_Calib_Pos_Done := FALSE;
END_IF

//================================================
// Reset / Disable
//================================================

IF Reset OR NOT Enable THEN
    State := 0;
    StartOld := FALSE;
    Busy := FALSE;
    DoneAll := FALSE;
    Error := FALSE;
    ErrorID := 0;
    CurrentIndex := 0;

    IF Hand_No = 1 THEN
        ARunP := FALSE;
    END_IF;

    IF Hand_No = 2 THEN
        BRunP := FALSE;
    END_IF;

    Trigger_RB := FALSE;
    Run_Calib_Pos_Done := FALSE;

    IF CameraID >= 1 AND CameraID <= GVL.C_MAX_VISION_CHANNELS THEN
        GVL.g_aVisionModbusControl[CameraID].RunCalib := FALSE;
        GVL.g_aVisionModbusControl[CameraID].CalibPosReady := FALSE;
    END_IF;

    tTimeout(IN := FALSE);
    t_Delay_Trigger.IN := FALSE;

    Trigger_Done_Old := FALSE;
    Calib_Done_Old := FALSE;

    RETURN;
END_IF;


//================================================
// Timeout
//================================================
// tTimeout(
//     IN := Busy AND (State <> 0) AND (State <> 100) AND NOT Error,
//     PT := TimeoutTime
// );
// 
// IF tTimeout.Q THEN
//     Error := TRUE;
//     ErrorID := 10; // timeout
//     State := 900;
// END_IF;


//================================================
// Motion Error
//================================================
IF (A_Error AND Hand_No = 1) THEN
    Error := TRUE;
    ErrorID := 20; // motion error
    State := 900;
END_IF;
IF (B_Error AND Hand_No = 2) THEN
    Error := TRUE;
    ErrorID := 20; // motion error
    State := 900;
END_IF;

//================================================
// State machine
//================================================
CASE State OF

    0: // IDLE
		Busy := FALSE;
		DoneAll := FALSE;
		Error := FALSE;
		ErrorID := 0;
	
		IF Start AND NOT StartOld THEN
	
			IF CameraID < 1 OR CameraID > GVL.C_MAX_VISION_CHANNELS THEN
				Error := TRUE;
				ErrorID := 3; // CameraID sai
				State := 900;
	
			ELSIF PointCount <= 0 THEN
				Error := TRUE;
				ErrorID := 1; // PointCount sai
				State := 900;
	
			ELSIF PointCount > 12 THEN
				Error := TRUE;
				ErrorID := 2; // Qua 12 diem calib
				State := 900;
	
			ELSE
				CurrentIndex := 1;
				Busy := TRUE;
				DoneAll := FALSE;
				Run_Calib_Pos_Done := FALSE;
	
				IF NOT Run_No_Trigger THEN
					GVL.g_aVisionModbusControl[CameraID].RunCalib := TRUE;
					GVL.g_aVisionModbusControl[CameraID].CalibPosReady := FALSE;
					GVL.g_aVisionModbusControl[CameraID].CalibPointCount := INT_TO_UINT(PointCount);
	
					GVL.g_aVisionCommand[CameraID].CameraID := CameraID;
					GVL.g_aVisionCommand[CameraID].Application := E_VisionApplication.VIS_APP_CALIBRATION;
					GVL.g_aVisionCommand[CameraID].Execute := FALSE;
					GVL.g_aVisionCommand[CameraID].Abort := FALSE;
					GVL.g_aVisionCommand[CameraID].Reset := FALSE;
				END_IF;
	
				State := 10;
			END_IF;
	
		END_IF;


    10: // LOAD POINT
		IF Run_Mode THEN
			Tmp_Delta := FC_CalcCalibPoint(Index := CurrentIndex, PointNo1 := PointNo1, NumberPoint_X := Nb_Point_X, NumberPoint_Y := Nb_Point_Y, Delta_X := Delta_X, Delta_Y := Delta_Y, Delta_A := Delta_A); 
			IF Hand_No = 1 THEN
				CurrentPoint_Run_A.c.X := GVL_1.DATA_RB_A.X_POS[PointNo1] + Tmp_Delta.X;
				CurrentPoint_Run_A.c.Y := GVL_1.DATA_RB_A.Y_POS[PointNo1] + Tmp_Delta.Y;
				CurrentPoint_Run_A.c.Z := GVL_1.DATA_RB_A.Z_POS[PointNo1] + Tmp_Delta.Z;
				CurrentPoint_Run_A.c.A := GVL_1.DATA_RB_A.R_POS[PointNo1] + Tmp_Delta.A;
			END_IF;
			IF Hand_No = 2 THEN
				CurrentPoint_Run_B.c.X := GVL_1.DATA_RB_B.X_POS[PointNo1] + Tmp_Delta.X;
				CurrentPoint_Run_B.c.Y := GVL_1.DATA_RB_B.Y_POS[PointNo1] + Tmp_Delta.Y;
				CurrentPoint_Run_B.c.Z := GVL_1.DATA_RB_B.Z_POS[PointNo1] + Tmp_Delta.Z;
				CurrentPoint_Run_B.c.A := GVL_1.DATA_RB_B.R_POS[PointNo1] + Tmp_Delta.A;
			END_IF;
		ELSE
			IF Hand_No = 1 THEN
				CurrentPoint_Run_A.c.X := GVL_1.DATA_RB_A.X_POS[PointNo1 + CurrentIndex - 1];
				CurrentPoint_Run_A.c.Y := GVL_1.DATA_RB_A.Y_POS[PointNo1 + CurrentIndex - 1];
				CurrentPoint_Run_A.c.Z := GVL_1.DATA_RB_A.Z_POS[PointNo1 + CurrentIndex - 1];
				CurrentPoint_Run_A.c.A := GVL_1.DATA_RB_A.R_POS[PointNo1 + CurrentIndex - 1];
			END_IF;
			IF Hand_No = 2 THEN
				CurrentPoint_Run_B.c.X := GVL_1.DATA_RB_B.X_POS[PointNo1 + CurrentIndex - 1];
				CurrentPoint_Run_B.c.Y := GVL_1.DATA_RB_B.Y_POS[PointNo1 + CurrentIndex - 1];
				CurrentPoint_Run_B.c.Z := GVL_1.DATA_RB_B.Z_POS[PointNo1 + CurrentIndex - 1];
				CurrentPoint_Run_B.c.A := GVL_1.DATA_RB_B.R_POS[PointNo1 + CurrentIndex - 1];
			END_IF;
		END_IF;
        State := 20;


    20: // SEND MOVE COMMAND
        //MoveCmd := TRUE; // xung 1 scan yêu cầu motion chạy điểm
		IF Hand_No = 1 AND NOT ARunP AND NOT A_Comp THEN
			ARunP := TRUE;
		END_IF;
		
		IF Hand_No = 2 AND NOT BRunP AND NOT B_Comp THEN
			BRunP := TRUE;
		END_IF;
		
        State := 30;


    30: // WAIT MOVE DONE + SAVE ACTUAL POSITION

		IF Hand_No = 1 AND A_Comp THEN
			ARunP := FALSE;
			A_Comp := FALSE;
	
			IF NOT Run_No_Trigger THEN
				GVL.g_aVisionModbusControl[CameraID].CalibrationPoints[CurrentIndex].X := TO_REAL(GVL.RB_A_.CUR_X);
				GVL.g_aVisionModbusControl[CameraID].CalibrationPoints[CurrentIndex].Y := TO_REAL(GVL.RB_A_.CUR_Y);
				GVL.g_aVisionModbusControl[CameraID].CalibrationPoints[CurrentIndex].Z := TO_REAL(GVL.RB_A_.CUR_Z);
				GVL.g_aVisionModbusControl[CameraID].CalibrationPoints[CurrentIndex].A := TO_REAL(GVL.RB_A_.CUR_R);
			END_IF;
	
			State := 40;
		END_IF;
	
		IF Hand_No = 2 AND B_Comp THEN
			BRunP := FALSE;
			B_Comp := FALSE;
	
			IF NOT Run_No_Trigger THEN
				GVL.g_aVisionModbusControl[CameraID].CalibrationPoints[CurrentIndex].X := TO_REAL(GVL.RB_B_.CUR_X);
				GVL.g_aVisionModbusControl[CameraID].CalibrationPoints[CurrentIndex].Y := TO_REAL(GVL.RB_B_.CUR_Y);
				GVL.g_aVisionModbusControl[CameraID].CalibrationPoints[CurrentIndex].Z := TO_REAL(GVL.RB_B_.CUR_Z);
				GVL.g_aVisionModbusControl[CameraID].CalibrationPoints[CurrentIndex].A := TO_REAL(GVL.RB_B_.CUR_R);
			END_IF;
	
			State := 40;
		END_IF;
	
	
	40: // DELAY BEFORE CAPTURE
		t_Delay_Trigger.IN := TRUE;
	
		IF t_Delay_Trigger.Q THEN
			t_Delay_Trigger.IN := FALSE;
	
			IF Run_No_Trigger THEN
				State := 60;
			ELSE
				State := 45;
			END_IF;
		END_IF;
	
	
	45: // WAIT OLD TRIGGER DONE = FALSE
		GVL.g_aVisionCommand[CameraID].Execute := FALSE;

		IF NOT GVL.g_aVisionModbusStatus[CameraID].TriggerDone THEN
			State := 50;
		END_IF;
	
	
	50: // TRIGGER CURRENT CALIB POINT
		GVL.g_aVisionCommand[CameraID].CameraID := CameraID;
		GVL.g_aVisionCommand[CameraID].Application := E_VisionApplication.VIS_APP_CALIBRATION;
		GVL.g_aVisionCommand[CameraID].Execute := TRUE;
	
		State := 55;
	
	
	55: // WAIT TRIGGER DONE
    IF GVL.g_aVisionModbusStatus[CameraID].CalibError THEN
        Error := TRUE;
        ErrorID := 41;
        State := 900;

    ELSIF GVL.g_aVisionModbusStatus[CameraID].Error THEN
        Error := TRUE;
        ErrorID := 42;
        State := 900;

    ELSIF GVL.g_aVisionModbusStatus[CameraID].TriggerDone THEN
        GVL.g_aVisionCommand[CameraID].Execute := FALSE;
        State := 60;
    END_IF;
	
	
	58: // WAIT VISION RELEASE TRIGGER DONE
		IF NOT GVL.g_aVisionModbusStatus[CameraID].TriggerDone THEN
			State := 60;
		END_IF;
	
	
	60: // NEXT POINT / ALL POINTS READY
		t_Delay_Trigger.IN := FALSE;
	
		IF CurrentIndex >= PointCount THEN
			Run_Calib_Pos_Done := TRUE;
	
			IF Run_No_Trigger THEN
				Busy := FALSE;
				DoneAll := TRUE;
				State := 100;
			ELSE
				GVL.g_aVisionModbusControl[CameraID].CalibPosReady := TRUE;
				State := 70;
			END_IF;
	
		ELSE
			CurrentIndex := CurrentIndex + 1;
			State := 10;
		END_IF;
	
	
	70: // WAIT VISION CALIBRATION CALCULATION DONE
		IF GVL.g_aVisionModbusStatus[CameraID].CalibError THEN
			Error := TRUE;
			ErrorID := 43;
			State := 900;
	
		ELSIF GVL.g_aVisionModbusStatus[CameraID].Error THEN
			Error := TRUE;
			ErrorID := 44;
			State := 900;
	
		ELSIF GVL.g_aVisionModbusStatus[CameraID].CalibDone THEN
			GVL.g_aVisionModbusControl[CameraID].CalibPosReady := FALSE;
			GVL.g_aVisionModbusControl[CameraID].RunCalib := FALSE;
	
			Run_Calib_Pos_Done := FALSE;
			Busy := FALSE;
			DoneAll := TRUE;
	
			State := 100;
		END_IF;
	
	
	100: // DONE
		Busy := FALSE;
	
		IF NOT Start THEN
			State := 0;
		END_IF;
	
	900: // ERROR
		Busy := FALSE;
	
		Trigger_RB := FALSE;
		Run_Calib_Pos_Done := FALSE;
	
		t_Delay_Trigger.IN := FALSE;
	
		IF CameraID >= 1 AND CameraID <= GVL.C_MAX_VISION_CHANNELS THEN
			GVL.g_aVisionModbusControl[CameraID].RunCalib := FALSE;
			GVL.g_aVisionModbusControl[CameraID].CalibPosReady := FALSE;
		END_IF;
	
		IF Hand_No = 1 THEN
			ARunP := FALSE;
		END_IF;
	
		IF Hand_No = 2 THEN
			BRunP := FALSE;
		END_IF;

END_CASE;


//================================================
// Save old signals for edge detect
//================================================
StartOld := Start;
// Trigger_Done_Old := Triger_RB_Done;
// Calib_Done_Old := Calib_Done;

END_FUNCTION_BLOCK

// Just_Motion_Control_x86_64_Linux_SM_WV/Application/FC_/FC_CalcCalibPoint
FUNCTION FC_CalcCalibPoint  : ST_POS
VAR_INPUT
	Index  : INT; // bắt đầu từ 1
	PointNo1 : INT; // Diem calib dau tien
	NumberPoint_X : INT;
	NumberPoint_Y : INT;
	Delta_X : REAL;
	Delta_Y : REAL;
	Delta_A : REAL;
END_VAR
VAR
	idx0 : INT;
    ix   : INT;
    iy   : INT;
END_VAR

idx0 := Index - 1;

ix := idx0 MOD NumberPoint_X;
iy := idx0 / NumberPoint_X;

FC_CalcCalibPoint.X := INT_TO_LREAL(ix) * (Delta_X/100);
FC_CalcCalibPoint.Y := INT_TO_LREAL(iy) * (Delta_Y/100);
FC_CalcCalibPoint.Z := 0;
FC_CalcCalibPoint.A := INT_TO_LREAL(idx0) * (Delta_A/100);

END_FUNCTION

// Just_Motion_Control_x86_64_Linux_SM_WV/Application/FB_/FB_TriggerVS
FUNCTION_BLOCK FB_TriggerVS
VAR_INPUT
    Enable : BOOL;
    Start : BOOL;

    CameraID : UINT;
    JobID : UINT;
    Application : E_VisionApplication;

    count_Vs_Align_max : INT;
    T_Delay_Trigger_time : INT;

    Trigger_Again : BOOL;
    Pass_Triger_VS_NG : BOOL;
    Mode_ByPass_VS : BOOL;
END_VAR

VAR_OUTPUT
    Busy : BOOL;
    DoneAll : BOOL;
    Error : BOOL;
    ErrorID : INT;

    CurrentTriggerID : UDINT;
END_VAR

VAR
    State : INT;
    StartOld : BOOL;

    count_Vs_Align : INT;

    t_Delay_Trigger : TON;
    xDelayTrigger : BOOL;

    RTrig_Enable : R_TRIG;

    udiTriggerCounter : UDINT;
END_VAR

//=============================================================================
// FB_TriggerVS
// Trigger Vision + chờ TriggerDone.
// T_Delay_Trigger_time được dùng làm TIMEOUT tối đa.
//=============================================================================


//=============================================================================
// ENABLE RISING EDGE
//=============================================================================
RTrig_Enable(CLK := Enable);

IF RTrig_Enable.Q THEN
    State := 0;
    StartOld := FALSE;

    Busy := FALSE;
    DoneAll := FALSE;
    Error := FALSE;
    ErrorID := 0;

    count_Vs_Align := 0;
    xDelayTrigger := FALSE;

    IF CameraID >= 1 AND CameraID <= GVL.C_MAX_VISION_CHANNELS THEN
        GVL.g_aVisionCommand[CameraID].Execute := FALSE;
        GVL.g_aVisionCommand[CameraID].Abort := FALSE;
        GVL.g_aVisionCommand[CameraID].Reset := FALSE;
    END_IF;
END_IF;


//=============================================================================
// DISABLE
//=============================================================================
IF NOT Enable THEN
    State := 0;
    StartOld := FALSE;

    Busy := FALSE;
    DoneAll := FALSE;
    Error := FALSE;
    ErrorID := 0;

    count_Vs_Align := 0;
    xDelayTrigger := FALSE;

    IF CameraID >= 1 AND CameraID <= GVL.C_MAX_VISION_CHANNELS THEN
        GVL.g_aVisionCommand[CameraID].Execute := FALSE;
    END_IF;

    // Reset TON ngay khi Disable.
    t_Delay_Trigger(IN := FALSE, PT := TO_TIME(T_Delay_Trigger_time) * 100);

    RETURN;
END_IF;


//=============================================================================
// STATE MACHINE
//=============================================================================
CASE State OF

    //-------------------------------------------------------------------------
    // STATE 0 - IDLE
    //-------------------------------------------------------------------------
    0:
        Busy := FALSE;
        DoneAll := FALSE;
        Error := FALSE;
        ErrorID := 0;

        count_Vs_Align := 0;
        xDelayTrigger := FALSE;

        IF Start AND NOT StartOld THEN

            IF CameraID < 1 OR CameraID > GVL.C_MAX_VISION_CHANNELS THEN
                Error := TRUE;
                ErrorID := 1;
                State := 900;

            ELSIF Mode_ByPass_VS THEN
                State := 30;

            ELSE
                Busy := TRUE;
                State := 5;
            END_IF;

        END_IF;


    //-------------------------------------------------------------------------
    // STATE 5 - PREPARE TRIGGER
    //
    // Hạ Execute và reset Timer trước khi phát Trigger mới.
    // Nếu TriggerDone cũ vẫn TRUE thì chờ nó hạ.
    //-------------------------------------------------------------------------
    5:
        GVL.g_aVisionCommand[CameraID].Execute := FALSE;
        xDelayTrigger := FALSE;

        IF NOT GVL.g_aVisionModbusStatus[CameraID].TriggerDone THEN
            State := 10;
        END_IF;


    //-------------------------------------------------------------------------
    // STATE 10 - SEND TRIGGER
    //
    // Tạo TriggerID mới và bật Execute.
    //-------------------------------------------------------------------------
    10:
        udiTriggerCounter := udiTriggerCounter + 1;

        IF udiTriggerCounter = 0 THEN
            udiTriggerCounter := 1;
        END_IF;

        CurrentTriggerID := udiTriggerCounter;

        GVL.g_aVisionCommand[CameraID].CameraID := CameraID;
        GVL.g_aVisionCommand[CameraID].JobID := JobID;
        GVL.g_aVisionCommand[CameraID].Application := Application;
        GVL.g_aVisionCommand[CameraID].TriggerID := CurrentTriggerID;

        GVL.g_aVisionCommand[CameraID].Abort := FALSE;
        GVL.g_aVisionCommand[CameraID].Reset := FALSE;
        GVL.g_aVisionCommand[CameraID].Execute := TRUE;

        // Bắt đầu Timeout từ Trigger này.
        xDelayTrigger := TRUE;

        State := 20;


    //-------------------------------------------------------------------------
    // STATE 20 - WAIT TRIGGER DONE
    //
    // Ưu tiên TriggerDone.
    // Chỉ Timeout nếu hết thời gian mà chưa nhận TriggerDone.
    //-------------------------------------------------------------------------
    20:
        GVL.g_aVisionCommand[CameraID].Execute := TRUE;

        IF GVL.g_aVisionModbusStatus[CameraID].TriggerDone THEN
            GVL.g_aVisionCommand[CameraID].Execute := FALSE;
            xDelayTrigger := FALSE;

            State := 30;

        ELSIF t_Delay_Trigger.Q THEN
            GVL.g_aVisionCommand[CameraID].Execute := FALSE;
            xDelayTrigger := FALSE;

            count_Vs_Align := count_Vs_Align + 1;

            IF count_Vs_Align < count_Vs_Align_max THEN
                State := 5;
            ELSE
                Error := TRUE;
                ErrorID := 2;
                State := 900;
            END_IF;
        END_IF;


    //-------------------------------------------------------------------------
    // STATE 30 - TRIGGER DONE
    //
    // Chỉ có nghĩa Trigger handshake đã nhận TriggerDone.
    // Result Vision sẽ do FB_VisionWaitResult xử lý.
    //-------------------------------------------------------------------------
    30:
        IF CameraID >= 1 AND CameraID <= GVL.C_MAX_VISION_CHANNELS THEN
            GVL.g_aVisionCommand[CameraID].Execute := FALSE;
        END_IF;

        xDelayTrigger := FALSE;

        Busy := FALSE;
        DoneAll := TRUE;
        Error := FALSE;
        ErrorID := 0;

        IF NOT Start THEN
            State := 0;
        END_IF;


    //-------------------------------------------------------------------------
    // STATE 900 - ERROR
    //
    // ErrorID:
    // 1 = CameraID không hợp lệ.
    // 2 = Trigger Timeout quá số lần cho phép.
    //-------------------------------------------------------------------------
    900: // ERROR
		IF CameraID >= 1 AND CameraID <= GVL.C_MAX_VISION_CHANNELS THEN
			GVL.g_aVisionCommand[CameraID].Execute := FALSE;
		END_IF;
	
		xDelayTrigger := FALSE;
	
		Busy := FALSE;
		DoneAll := FALSE;
	
		// Nếu người dùng yêu cầu Trigger lại ngay khi Start vẫn còn giữ.
		IF Trigger_Again THEN
			Error := FALSE;
			ErrorID := 0;
			count_Vs_Align := 0;
	
			State := 5;
	
		// Khi bên gọi nhả Start thì kết thúc chu trình lỗi,
		// reset FB để sẵn sàng cho lần Start tiếp theo.
		ELSIF NOT Start THEN
			Error := FALSE;
			ErrorID := 0;
			count_Vs_Align := 0;
	
			State := 0;
		END_IF;

END_CASE;


//=============================================================================
// TIMER
//
// ĐẶT SAU STATE MACHINE.
// Như vậy xDelayTrigger vừa được thay đổi trong State hiện tại sẽ tác động
// ngay vào TON trong chính scan này.
//=============================================================================
t_Delay_Trigger(
    IN := xDelayTrigger,
    PT := TO_TIME(T_Delay_Trigger_time) * 100
);


//=============================================================================
// SAVE OLD SIGNAL
//=============================================================================
StartOld := Start;

END_FUNCTION_BLOCK

// Just_Motion_Control_x86_64_Linux_SM_WV/Application/FB_/Vision/FB_VisionWaitResult
FUNCTION_BLOCK FB_VisionWaitResult
VAR_INPUT
    Enable : BOOL;                              // Cho phép FB hoạt động.
    Start : BOOL;                               // Cạnh lên bắt đầu chờ Result từ Vision.

    CameraID : UINT;                            // ID Camera cần lấy Result: 1..C_MAX_VISION_CHANNELS.
    ExpectedTriggerID : UDINT;                  // TriggerID PLC đang chờ. Phải trùng TriggerID Vision trả về.
    ExpectedJobID : UINT;                       // JobID mong đợi. Dùng để tránh nhận nhầm kết quả của Job khác.
    ExpectedApplication : E_VisionApplication; // Loại ứng dụng mong đợi: ALIGN, PICK_POSITION...
END_VAR

VAR_OUTPUT
    Busy : BOOL;                                // TRUE khi FB đang chờ/xử lý Result.
    Done : BOOL;                                // TRUE khi đã nhận và copy xong Result đúng yêu cầu.
    Error : BOOL;                               // TRUE khi có lỗi trong quá trình chờ Result.
    ErrorID : INT;                              // Mã lỗi nội bộ của FB.

    ResultValid : BOOL;                         // TRUE khi PosResult phía Vision báo tọa độ hợp lệ.
    ResultOK : BOOL;                            // TRUE khi ResultValid và ResultStatus = VIS_RESULT_OK.

    ResultX : REAL;                             // Tọa độ/Offset X Vision trả về.
    ResultY : REAL;                             // Tọa độ/Offset Y Vision trả về.
    ResultZ : REAL;                             // Tọa độ/Offset Z Vision trả về.
    ResultA : REAL;                             // Góc A Vision trả về.
    ResultScore : REAL;                         // Điểm nhận dạng của Vision.
    ResultFeatureID : UINT;                     // ID Feature/Pattern Vision nhận dạng được.

    ResultStatus : E_VisionResultStatus;        // Trạng thái kết quả: OK, NG, NOT_FOUND, LOW_SCORE...
    ResultCode : UINT;                          // Mã kết quả do Vision trả về.
    VisionErrorCode : UINT;                     // Mã lỗi do Vision trả về.

    ReceivedTriggerID : UDINT;                  // TriggerID thực tế của Result đã được FB nhận.
END_VAR

VAR
    State : INT;                                // State machine nội bộ của FB.
    StartOld : BOOL;                            // Lưu Start scan trước để bắt cạnh lên.

    tResultTimeout : TON;                       // Timer giới hạn thời gian chờ Vision trả Result.
    xResultTimeout : BOOL;                      // Enable cho timer chờ Result.
END_VAR

//=============================================================================
// FB_VisionWaitResult
// Chức năng:
// - Chờ Result đã được FB_VisionModbusDriver decode.
// - Chỉ nhận Result đúng TriggerID + JobID + Application.
// - Copy dữ liệu X/Y/Z/A/Score ra Output.
// - KHÔNG điều khiển AckResult tại đây.
//   AckResult thuộc quyền quản lý của FB_VisionModbusDriver.
//=============================================================================


//=============================================================================
// 1. RESULT TIMEOUT
// Dùng thời gian timeout đã cấu hình riêng cho từng Camera.
//=============================================================================
IF CameraID >= 1 AND CameraID <= GVL.C_MAX_VISION_CHANNELS THEN
    tResultTimeout(IN := xResultTimeout, PT := TO_TIME(GVL.g_aVisionConfig[CameraID].ResultTimeout *100));
ELSE
    tResultTimeout(IN := FALSE);
END_IF;


//=============================================================================
// 2. DISABLE
// Khi FB bị Disable: đưa toàn bộ trạng thái nội bộ và Output về mặc định.
// Không can thiệp vào AckResult vì handshake Modbus thuộc Driver.
//=============================================================================
IF NOT Enable THEN
    State := 0;
    StartOld := FALSE;

    Busy := FALSE;
    Done := FALSE;
    Error := FALSE;
    ErrorID := 0;

    ResultValid := FALSE;
    ResultOK := FALSE;

    ResultX := 0.0;
    ResultY := 0.0;
    ResultZ := 0.0;
    ResultA := 0.0;
    ResultScore := 0.0;
    ResultFeatureID := 0;

    ResultStatus := E_VisionResultStatus.VIS_RESULT_NONE;
    ResultCode := 0;
    VisionErrorCode := 0;
    ReceivedTriggerID := 0;

    xResultTimeout := FALSE;

    RETURN;
END_IF;


//=============================================================================
// 3. STATE MACHINE
//=============================================================================
CASE State OF

    //-------------------------------------------------------------------------
    // STATE 0 - IDLE
    // Chờ cạnh lên của Start.
    // Kiểm tra CameraID và ExpectedTriggerID trước khi bắt đầu chờ Result.
    //-------------------------------------------------------------------------
    0:
        Busy := FALSE;
        Done := FALSE;
        Error := FALSE;
        ErrorID := 0;

        ResultValid := FALSE;
        ResultOK := FALSE;

        xResultTimeout := FALSE;

        IF Start AND NOT StartOld THEN

            // CameraID ngoài phạm vi cấu hình.
            IF CameraID < 1 OR CameraID > GVL.C_MAX_VISION_CHANNELS THEN
                Error := TRUE;
                ErrorID := 1;
                State := 900;

            // TriggerID = 0 không được coi là một Trigger hợp lệ.
            ELSIF ExpectedTriggerID = 0 THEN
                Error := TRUE;
                ErrorID := 2;
                State := 900;

            ELSE
                // Bắt đầu chờ Result tương ứng với Trigger đã gửi.
                Busy := TRUE;
                xResultTimeout := TRUE;
                State := 10;
            END_IF;

        END_IF;


    //-------------------------------------------------------------------------
    // STATE 10 - WAIT MATCHING RESULT
    // Chờ Driver decode được một Result hoàn chỉnh.
    //
    // Điều kiện nhận Result:
    // 1. Header.Valid = TRUE.
    // 2. TriggerID đúng Trigger đang chờ.
    // 3. JobID đúng Job đang chạy.
    // 4. Application đúng loại ứng dụng đang chạy.
    //
    // Result cũ có TriggerID khác sẽ bị bỏ qua và tiếp tục chờ.
    //-------------------------------------------------------------------------
    10:
        // Vision/Modbus báo lỗi.
        IF GVL.g_aVisionModbusStatus[CameraID].Error THEN
            Error := TRUE;
            ErrorID := 10;
            xResultTimeout := FALSE;
            State := 900;

        // Quá thời gian chờ Vision trả Result.
        ELSIF tResultTimeout.Q THEN
            Error := TRUE;
            ErrorID := 11;
            xResultTimeout := FALSE;
            State := 900;

        // Driver đã decode được một Result hoàn chỉnh.
        ELSIF GVL.g_aVisionResult[CameraID].Header.Valid THEN

            // Chỉ xử lý Result thuộc đúng Trigger hiện tại.
            IF GVL.g_aVisionResult[CameraID].Header.TriggerID = ExpectedTriggerID THEN

                // Trigger đúng nhưng JobID không đúng.
                IF GVL.g_aVisionResult[CameraID].Header.JobID <> ExpectedJobID THEN
                    Error := TRUE;
                    ErrorID := 12;
                    xResultTimeout := FALSE;
                    State := 900;

                // Trigger + Job đúng nhưng Application không đúng.
                ELSIF GVL.g_aVisionResult[CameraID].Header.Application <> ExpectedApplication THEN
                    Error := TRUE;
                    ErrorID := 13;
                    xResultTimeout := FALSE;
                    State := 900;

                ELSE
                    // Result hoàn toàn đúng Request đang chờ.
                    State := 20;
                END_IF;

            END_IF;
        END_IF;


    //-------------------------------------------------------------------------
    // STATE 20 - COPY RESULT
    // Result đã được xác nhận đúng TriggerID + JobID + Application.
    // Copy dữ liệu từ vùng Result chung sang Output riêng của FB.
    //-------------------------------------------------------------------------
    20:
        xResultTimeout := FALSE;

        // Lưu TriggerID thực tế đã nhận để theo dõi/debug.
        ReceivedTriggerID := GVL.g_aVisionResult[CameraID].Header.TriggerID;

        // Copy Header Result.
        ResultStatus := GVL.g_aVisionResult[CameraID].Header.ResultStatus;
        ResultCode := GVL.g_aVisionResult[CameraID].Header.ResultCode;
        VisionErrorCode := GVL.g_aVisionResult[CameraID].Header.ErrorCode;

        // Copy trạng thái Position Result.
        ResultValid := GVL.g_aVisionResult[CameraID].PosResult.Valid;

        // Copy tọa độ/Offset Vision đã decode.
        ResultX := GVL.g_aVisionResult[CameraID].PosResult.Pos.X;
        ResultY := GVL.g_aVisionResult[CameraID].PosResult.Pos.Y;
        ResultZ := GVL.g_aVisionResult[CameraID].PosResult.Pos.Z;
        ResultA := GVL.g_aVisionResult[CameraID].PosResult.Pos.A;

        // Copy thông tin nhận dạng.
        ResultScore := GVL.g_aVisionResult[CameraID].PosResult.Score;
        ResultFeatureID := GVL.g_aVisionResult[CameraID].PosResult.FeatureID;

        // Result chỉ được coi là OK khi:
        // - Position hợp lệ.
        // - Vision trả trạng thái VIS_RESULT_OK.
        ResultOK := ResultValid AND (ResultStatus = E_VisionResultStatus.VIS_RESULT_OK);

        Busy := FALSE;
        Done := TRUE;

        State := 30;


    //-------------------------------------------------------------------------
    // STATE 30 - DONE
    // Giữ Done = TRUE cho đến khi chương trình gọi FB nhả Start.
    //-------------------------------------------------------------------------
    30:
        Busy := FALSE;
        Done := TRUE;

        IF NOT Start THEN
            State := 0;
        END_IF;


    //-------------------------------------------------------------------------
    // STATE 900 - ERROR
    // Giữ trạng thái Error cho đến khi Start được nhả.
    // ErrorID cho biết nguyên nhân lỗi cụ thể.
    //-------------------------------------------------------------------------
    900:
        Busy := FALSE;
        Done := FALSE;
        xResultTimeout := FALSE;

        IF NOT Start THEN
            State := 0;
        END_IF;

END_CASE;


//=============================================================================
// 4. SAVE OLD SIGNAL
// Lưu Start cuối scan để phát hiện cạnh lên ở scan tiếp theo.
//=============================================================================
StartOld := Start;

END_FUNCTION_BLOCK

// Just_Motion_Control_x86_64_Linux_SM_WV/Application/FB_/Modbus/FB_VisionModbusDriver
FUNCTION_BLOCK FB_VisionModbusDriver
VAR_INPUT
    Enable : BOOL;
    Reset : BOOL;
    Config : ST_VISION_CONFIG;
    Command : ST_VISION_COMMAND;
END_VAR

VAR_IN_OUT
    ModbusControl : ST_VISION_MODBUS_CONTROL;
    ChannelStatus : ST_VISION_CHANNEL_STATUS;
    ModbusStatus : ST_VISION_MODBUS_STATUS;
    VisionResult : ST_VISION_RESULT;
    Registers : ARRAY[0..1999] OF WORD;
END_VAR

VAR_OUTPUT
    Active : BOOL;
    Error : BOOL;
    ErrorID : UDINT;
END_VAR

VAR
    uiBase : UINT;
    uiR2V : UINT;
    uiV2R : UINT;
    uiData : UINT;
    uiMulti : UINT;
    wControl : WORD;
    wStatus : WORD;
    wObjectInfo : WORD;
    diRaw : DINT;
    udiTriggerID : UDINT;
    uiPoint : UINT;
    uiRecord : UINT;
    uiGlobalObject : UINT;
    uiBlockIndex : UINT;
    uiBlockDataCount : UINT;
    rPositionScale : REAL;
    rAngleScale : REAL;
    rScoreScale : REAL;
    udiLastResultTriggerID : UDINT;
    udiLastBlockTriggerID : UDINT;
    uiLastDecodedBlock : UINT;
    xLastHeartbeat : BOOL;
    xHeartbeatToggle : BOOL;
    tHeartbeatTimeout : TON;
END_VAR

// //=============================================================================
// // RESET / DISABLE
// //=============================================================================
// IF Reset OR NOT Enable THEN
//     Active := FALSE;
//     Error := FALSE;
//     ErrorID := 0;
// 
//     //---------------------------------------------------------------------
//     // XÓA BỘ NHỚ TRANSACTION CŨ.
//     //---------------------------------------------------------------------
//     udiLastResultTriggerID := 0;
//     udiLastBlockTriggerID := 0;
//     uiLastDecodedBlock := 0;
// 
//     //---------------------------------------------------------------------
//     // XÓA RESULT CŨ.
//     //---------------------------------------------------------------------
//     VisionResult.Header.Valid := FALSE;
//     VisionResult.Header.TriggerID := 0;
// 
//     VisionResult.TrackObjectResult.Valid := FALSE;
//     VisionResult.TrackObjectResult.ObjectCount := 0;
// 
//     //---------------------------------------------------------------------
//     // XÓA HANDSHAKE CŨ.
//     //---------------------------------------------------------------------
//     ModbusControl.AckBlock := FALSE;
//     ModbusControl.AckResult := FALSE;
//     ModbusControl.AckBlockIndex := 0;
//     ModbusControl.RequestBlockIndex := 0;
//     RETURN;
// END_IF;

//=============================================================================
// MEMORY BASE
//=============================================================================
uiBase := Config.BaseAddress;
uiR2V := uiBase + Config.CommandOffset;
uiV2R := uiBase + Config.StatusOffset;
uiData := uiBase + Config.DataOffset;
uiMulti := uiBase + 132;

//=============================================================================
// VALIDATE ADDRESS
//=============================================================================
IF uiR2V + 99 > 1199 OR uiV2R + 199 > 1199 THEN
    Error := TRUE;
    ErrorID := 9251;
    RETURN;
END_IF;


//=============================================================================
// RESET
//-----------------------------------------------------------------------------
// Quan trọng:
// Phải gửi Reset sang Vision TRƯỚC khi RETURN.
//=============================================================================
IF Reset THEN

    //---------------------------------------------------------------------
    // 1. GỬI RESET SANG VISION
    //---------------------------------------------------------------------
    wControl := WORD#0;
    wControl.0 := TRUE;          // Heartbeat.
    wControl.6 := TRUE;          // RESET.
    Registers[uiR2V + 0] := wControl;

    //---------------------------------------------------------------------
    // 2. RESET INTERNAL TRANSACTION
    //---------------------------------------------------------------------
    Active := FALSE;
    Error := FALSE;
    ErrorID := 0;

    udiLastResultTriggerID := 0;
    udiLastBlockTriggerID := 0;
    uiLastDecodedBlock := 0;

    xLastHeartbeat := FALSE;
    xHeartbeatToggle := FALSE;

    //---------------------------------------------------------------------
    // 3. RESET RESULT
    //---------------------------------------------------------------------
    VisionResult.Header.Valid := FALSE;
    VisionResult.Header.TriggerID := 0;
    VisionResult.Header.JobID := 0;
    VisionResult.Header.ResultCode := 0;
    VisionResult.Header.ErrorCode := 0;
    VisionResult.Header.DataCount := 0;
    VisionResult.Header.BlockCount := 0;
    VisionResult.Header.BlockIndex := 0;
    VisionResult.Header.BlockDataCount := 0;
    VisionResult.Header.CaptureConveyorPos := 0.0;

    VisionResult.TrackObjectResult.Valid := FALSE;
    VisionResult.TrackObjectResult.ObjectCount := 0;

    FOR uiRecord := 1 TO GVL.C_MAX_VISION_TRACK_OBJECTS_PER_FRAME DO
        VisionResult.TrackObjectResult.Objects[uiRecord].Valid := FALSE;
        VisionResult.TrackObjectResult.Objects[uiRecord].Pos.X := 0.0;
        VisionResult.TrackObjectResult.Objects[uiRecord].Pos.Y := 0.0;
        VisionResult.TrackObjectResult.Objects[uiRecord].Pos.Z := 0.0;
        VisionResult.TrackObjectResult.Objects[uiRecord].Pos.A := 0.0;
        VisionResult.TrackObjectResult.Objects[uiRecord].Score := 0.0;
        VisionResult.TrackObjectResult.Objects[uiRecord].ProductClassID := 0;
        VisionResult.TrackObjectResult.Objects[uiRecord].FeatureID := 0;
    END_FOR;

    //---------------------------------------------------------------------
    // 4. RESET HANDSHAKE
    //---------------------------------------------------------------------
    ModbusControl.AckBlock := FALSE;
    ModbusControl.AckResult := FALSE;
    ModbusControl.AckBlockIndex := 0;
    ModbusControl.RequestBlockIndex := 0;

    //---------------------------------------------------------------------
    // 5. RESET MODBUS STATUS
    //---------------------------------------------------------------------
    ModbusStatus.HeartBeat := FALSE;
    ModbusStatus.TriggerDone := FALSE;
    ModbusStatus.CalibDone := FALSE;
    ModbusStatus.ResultReady := FALSE;
    ModbusStatus.Busy := FALSE;
    ModbusStatus.Run1Slot := FALSE;
    ModbusStatus.BlockReady := FALSE;
    ModbusStatus.Error := FALSE;
    ModbusStatus.CalibBusy := FALSE;
    ModbusStatus.CalibError := FALSE;
    ModbusStatus.BlockIndex := 0;
    ModbusStatus.BlockDataCount := 0;

